   1:L PR[91] R[100]mm/sec CNT100;
   1:  PR[91,1] = PR[90,1] + -29.183;
   1:  PR[91,2] = PR[90,2] + 14.555;
   1:  PR[91,3] = PR[90,3] + 10.199;
   1:L PR[91] R[100]mm/sec CNT100;
   1:  PR[91,1] = PR[90,1] + -29.870;
   1:  PR[91,2] = PR[90,2] + 14.078;
   1:  PR[91,3] = PR[90,3] + 10.201;
   1:L PR[91] R[100]mm/sec CNT100;
   1:  PR[91,1] = PR[90,1] + -30.532;
   1:  PR[91,2] = PR[90,2] + 13.568;
   1:  PR[91,3] = PR[90,3] + 10.206;
   1:L PR[91] R[100]mm/sec CNT100;
   1:  PR[91,1] = PR[90,1] + -31.168;
   1:  PR[91,2] = PR[90,2] + 13.026;
   1:  PR[91,3] = PR[90,3] + 10.211;
   1:L PR[91] R[100]mm/sec CNT100;
   1:  PR[91,1] = PR[90,1] + -31.777;
   1:  PR[91,2] = PR[90,2] + 12.454;
   1:  PR[91,3] = PR[90,3] + 10.217;
   1:L PR[91] R[100]mm/sec CNT100;
   1:  PR[91,1] = PR[90,1] + -32.357;
   1:  PR[91,2] = PR[90,2] + 11.852;
   1:  PR[91,3] = PR[90,3] + 10.222;
   1:L PR[91] R[100]mm/sec CNT100;
   1:  PR[91,1] = PR[90,1] + -32.907;
   1:  PR[91,2] = PR[90,2] + 11.222;
   1:  PR[91,3] = PR[90,3] + 10.227;
   1:L PR[91] R[100]mm/sec CNT100;
   1:  PR[91,1] = PR[90,1] + -33.426;
   1:  PR[91,2] = PR[90,2] + 10.565;
   1:  PR[91,3] = PR[90,3] + 10.232;
   1:L PR[91] R[100]mm/sec CNT100;
   1:  PR[91,1] = PR[90,1] + -33.911;
   1:  PR[91,2] = PR[90,2] + 9.884;
   1:  PR[91,3] = PR[90,3] + 10.237;
   1:L PR[91] R[100]mm/sec CNT100;
   1:  PR[91,1] = PR[90,1] + -34.362;
   1:  PR[91,2] = PR[90,2] + 9.178;
   1:  PR[91,3] = PR[90,3] + 10.243;
   1:L PR[91] R[100]mm/sec CNT100;
   1:  PR[91,1] = PR[90,1] + -34.778;
   1:  PR[91,2] = PR[90,2] + 8.451;
   1:  PR[91,3] = PR[90,3] + 10.248;
   1:L PR[91] R[100]mm/sec CNT100;
   1:  PR[91,1] = PR[90,1] + -35.158;
   1:  PR[91,2] = PR[90,2] + 7.705;
   1:  PR[91,3] = PR[90,3] + 10.253;
   1:L PR[91] R[100]mm/sec CNT100;
   1:  PR[91,1] = PR[90,1] + -35.500;
   1:  PR[91,2] = PR[90,2] + 6.942;
   1:  PR[91,3] = PR[90,3] + 10.258;
   1:L PR[91] R[100]mm/sec CNT100;
   1:  PR[91,1] = PR[90,1] + -35.805;
   1:  PR[91,2] = PR[90,2] + 6.164;
   1:  PR[91,3] = PR[90,3] + 10.263;
   1:L PR[91] R[100]mm/sec CNT100;
   1:  PR[91,1] = PR[90,1] + -36.070;
   1:  PR[91,2] = PR[90,2] + 5.374;
   1:  PR[91,3] = PR[90,3] + 10.269;
   1:L PR[91] R[100]mm/sec CNT100;
   1:  PR[91,1] = PR[90,1] + -36.295;
   1:  PR[91,2] = PR[90,2] + 4.572;
   1:  PR[91,3] = PR[90,3] + 10.274;
   1:L PR[91] R[100]mm/sec CNT100;
   1:  PR[91,1] = PR[90,1] + -36.480;
   1:  PR[91,2] = PR[90,2] + 3.761;
   1:  PR[91,3] = PR[90,3] + 10.279;
   1:L PR[91] R[100]mm/sec CNT100;
   1:  PR[91,1] = PR[90,1] + -36.625;
   1:  PR[91,2] = PR[90,2] + 2.940;
   1:  PR[91,3] = PR[90,3] + 10.284;
   1:L PR[91] R[100]mm/sec CNT100;
   1:  PR[91,1] = PR[90,1] + -36.728;
   1:  PR[91,2] = PR[90,2] + 2.111;
   1:  PR[91,3] = PR[90,3] + 10.289;
   1:L PR[91] R[100]mm/sec CNT100;
   1:  PR[91,1] = PR[90,1] + -36.791;
   1:  PR[91,2] = PR[90,2] + 1.273;
   1:  PR[91,3] = PR[90,3] + 10.295;
   1:L PR[91] R[100]mm/sec CNT100;
   1:  PR[91,1] = PR[90,1] + -36.812;
   1:  PR[91,2] = PR[90,2] + 0.428;
   1:  PR[91,3] = PR[90,3] + 10.300;
   1:L PR[91] R[100]mm/sec CNT100;
   1:  PR[91,1] = PR[90,1] + -36.791;
   1:  PR[91,2] = PR[90,2] + -0.418;
   1:  PR[91,3] = PR[90,3] + 10.305;
   1:L PR[91] R[100]mm/sec CNT100;
   1:  PR[91,1] = PR[90,1] + -36.728;
   1:  PR[91,2] = PR[90,2] + -1.256;
   1:  PR[91,3] = PR[90,3] + 10.310;
   1:L PR[91] R[100]mm/sec CNT100;
   1:  PR[91,1] = PR[90,1] + -36.625;
   1:  PR[91,2] = PR[90,2] + -2.085;
   1:  PR[91,3] = PR[90,3] + 10.316;
   1:L PR[91] R[100]mm/sec CNT100;
   1:  PR[91,1] = PR[90,1] + -36.480;
   1:  PR[91,2] = PR[90,2] + -2.906;
   1:  PR[91,3] = PR[90,3] + 10.321;
   1:L PR[91] R[100]mm/sec CNT100;
   1:  PR[91,1] = PR[90,1] + -36.295;
   1:  PR[91,2] = PR[90,2] + -3.717;
   1:  PR[91,3] = PR[90,3] + 10.326;
   1:L PR[91] R[100]mm/sec CNT100;
   1:  PR[91,1] = PR[90,1] + -36.070;
   1:  PR[91,2] = PR[90,2] + -4.519;
   1:  PR[91,3] = PR[90,3] + 10.331;
   1:L PR[91] R[100]mm/sec CNT100;
   1:  PR[91,1] = PR[90,1] + -35.805;
   1:  PR[91,2] = PR[90,2] + -5.309;
   1:  PR[91,3] = PR[90,3] + 10.336;
   1:L PR[91] R[100]mm/sec CNT100;
   1:  PR[91,1] = PR[90,1] + -35.500;
   1:  PR[91,2] = PR[90,2] + -6.087;
   1:  PR[91,3] = PR[90,3] + 10.341;
   1:L PR[91] R[100]mm/sec CNT100;
   1:  PR[91,1] = PR[90,1] + -35.158;
   1:  PR[91,2] = PR[90,2] + -6.850;
   1:  PR[91,3] = PR[90,3] + 10.347;
   1:L PR[91] R[100]mm/sec CNT100;
   1:  PR[91,1] = PR[90,1] + -34.778;
   1:  PR[91,2] = PR[90,2] + -7.596;
   1:  PR[91,3] = PR[90,3] + 10.352;
   1:L PR[91] R[100]mm/sec CNT100;
   1:  PR[91,1] = PR[90,1] + -34.362;
   1:  PR[91,2] = PR[90,2] + -8.323;
   1:  PR[91,3] = PR[90,3] + 10.357;
   1:L PR[91] R[100]mm/sec CNT100;
   1:  PR[91,1] = PR[90,1] + -33.911;
   1:  PR[91,2] = PR[90,2] + -9.028;
   1:  PR[91,3] = PR[90,3] + 10.362;
   1:L PR[91] R[100]mm/sec CNT100;
   1:  PR[91,1] = PR[90,1] + -33.426;
   1:  PR[91,2] = PR[90,2] + -9.710;
   1:  PR[91,3] = PR[90,3] + 10.367;
   1:L PR[91] R[100]mm/sec CNT100;
   1:  PR[91,1] = PR[90,1] + -32.907;
   1:  PR[91,2] = PR[90,2] + -10.367;
   1:  PR[91,3] = PR[90,3] + 10.373;
   1:L PR[91] R[100]mm/sec CNT100;
   1:  PR[91,1] = PR[90,1] + -32.357;
   1:  PR[91,2] = PR[90,2] + -10.997;
   1:  PR[91,3] = PR[90,3] + 10.378;
   1:L PR[91] R[100]mm/sec CNT100;
   1:  PR[91,1] = PR[90,1] + -31.777;
   1:  PR[91,2] = PR[90,2] + -11.599;
   1:  PR[91,3] = PR[90,3] + 10.383;
   1:L PR[91] R[100]mm/sec CNT100;
   1:  PR[91,1] = PR[90,1] + -31.168;
   1:  PR[91,2] = PR[90,2] + -12.171;
   1:  PR[91,3] = PR[90,3] + 10.388;
   1:L PR[91] R[100]mm/sec CNT100;
   1:  PR[91,1] = PR[90,1] + -30.532;
   1:  PR[91,2] = PR[90,2] + -12.713;
   1:  PR[91,3] = PR[90,3] + 10.393;
   1:L PR[91] R[100]mm/sec CNT100;
   1:  PR[91,1] = PR[90,1] + -29.869;
   1:  PR[91,2] = PR[90,2] + -13.223;
   1:  PR[91,3] = PR[90,3] + 10.399;
   1:L PR[91] R[100]mm/sec CNT100;
   1:  PR[91,1] = PR[90,1] + -29.571;
   1:  PR[91,2] = PR[90,2] + -13.432;
   1:  PR[91,3] = PR[90,3] + 10.404;
   1:L PR[91] R[100]mm/sec CNT100;
   1:  PR[91,1] = PR[90,1] + -29.184;
   1:  PR[91,2] = PR[90,2] + -13.699;
   1:  PR[91,3] = PR[90,3] + 10.406;
   1:L PR[91] R[100]mm/sec CNT100;
   1:  PR[91,1] = PR[90,1] + -28.475;
   1:  PR[91,2] = PR[90,2] + -14.142;
   1:  PR[91,3] = PR[90,3] + 10.409;
   1:L PR[91] R[100]mm/sec CNT100;
   1:  PR[91,1] = PR[90,1] + -27.746;
   1:  PR[91,2] = PR[90,2] + -14.550;
   1:  PR[91,3] = PR[90,3] + 10.414;
   1:L PR[91] R[100]mm/sec CNT100;
   1:  PR[91,1] = PR[90,1] + -27.316;
   1:  PR[91,2] = PR[90,2] + -14.765;
   1:  PR[91,3] = PR[90,3] + 10.419;
   1:L PR[91] R[100]mm/sec CNT100;
   1:  PR[91,1] = PR[90,1] + -26.999;
   1:  PR[91,2] = PR[90,2] + -14.921;
   1:  PR[91,3] = PR[90,3] + 10.422;
   1:L PR[91] R[100]mm/sec CNT100;
   1:  PR[91,1] = PR[90,1] + -26.234;
   1:  PR[91,2] = PR[90,2] + -15.256;
   1:  PR[91,3] = PR[90,3] + 10.425;
   1:L PR[91] R[100]mm/sec CNT100;
   1:  PR[91,1] = PR[90,1] + -25.453;
   1:  PR[91,2] = PR[90,2] + -15.554;
   1:  PR[91,3] = PR[90,3] + 10.430;
   1:L PR[91] R[100]mm/sec CNT100;
   1:  PR[91,1] = PR[90,1] + -24.883;
   1:  PR[91,2] = PR[90,2] + -15.741;
   1:  PR[91,3] = PR[90,3] + 10.435;
   1:L PR[91] R[100]mm/sec CNT100;
   1:  PR[91,1] = PR[90,1] + -23.854;
   1:  PR[91,2] = PR[90,2] + -16.033;
   1:  PR[91,3] = PR[90,3] + 10.439;
   1:L PR[91] R[100]mm/sec CNT100;
   1:  PR[91,1] = PR[90,1] + -23.043;
   1:  PR[91,2] = PR[90,2] + -16.213;
   1:  PR[91,3] = PR[90,3] + 10.445;
   1:L PR[91] R[100]mm/sec CNT100;
   1:  PR[91,1] = PR[90,1] + -22.223;
   1:  PR[91,2] = PR[90,2] + -16.354;
   1:  PR[91,3] = PR[90,3] + 10.451;
   1:L PR[91] R[100]mm/sec CNT100;
   1:  PR[91,1] = PR[90,1] + -21.397;
   1:  PR[91,2] = PR[90,2] + -16.455;
   1:  PR[91,3] = PR[90,3] + 10.456;
   1:L PR[91] R[100]mm/sec CNT100;
   1:  PR[91,1] = PR[90,1] + -20.560;
   1:  PR[91,2] = PR[90,2] + -16.517;
   1:  PR[91,3] = PR[90,3] + 10.461;
   1:L PR[91] R[100]mm/sec CNT100;
   1:  PR[91,1] = PR[90,1] + -19.711;
   1:  PR[91,2] = PR[90,2] + -16.538;
   1:  PR[91,3] = PR[90,3] + 10.466;
   1:L PR[91] R[100]mm/sec CNT100;
   1:  PR[91,1] = PR[90,1] + -18.860;
   1:  PR[91,2] = PR[90,2] + -16.518;
   1:  PR[91,3] = PR[90,3] + 10.471;
   1:L PR[91] R[100]mm/sec CNT100;
   1:  PR[91,1] = PR[90,1] + -18.010;
   1:  PR[91,2] = PR[90,2] + -16.456;
   1:  PR[91,3] = PR[90,3] + 10.477;
   1:L PR[91] R[100]mm/sec CNT100;
   1:  PR[91,1] = PR[90,1] + -17.397;
   1:  PR[91,2] = PR[90,2] + -16.381;
   1:  PR[91,3] = PR[90,3] + 10.482;
   1:L PR[91] R[100]mm/sec CNT100;
   1:  PR[91,1] = PR[90,1] + -16.320;
   1:  PR[91,2] = PR[90,2] + -16.206;
   1:  PR[91,3] = PR[90,3] + 10.486;
   1:L PR[91] R[100]mm/sec CNT100;
   1:  PR[91,1] = PR[90,1] + -15.489;
   1:  PR[91,2] = PR[90,2] + -16.020;
   1:  PR[91,3] = PR[90,3] + 10.493;
   1:L PR[91] R[100]mm/sec CNT100;
   1:  PR[91,1] = PR[90,1] + -15.048;
   1:  PR[91,2] = PR[90,2] + -15.900;
   1:  PR[91,3] = PR[90,3] + 10.498;
   1:L PR[91] R[100]mm/sec CNT100;
   1:  PR[91,1] = PR[90,1] + -14.666;
   1:  PR[91,2] = PR[90,2] + -15.793;
   1:  PR[91,3] = PR[90,3] + 10.501;
   1:L PR[91] R[100]mm/sec CNT100;
   1:  PR[91,1] = PR[90,1] + -13.853;
   1:  PR[91,2] = PR[90,2] + -15.525;
   1:  PR[91,3] = PR[90,3] + 10.503;
   1:L PR[91] R[100]mm/sec CNT100;
   1:  PR[91,1] = PR[90,1] + -13.057;
   1:  PR[91,2] = PR[90,2] + -15.217;
   1:  PR[91,3] = PR[90,3] + 10.509;
   1:L PR[91] R[100]mm/sec CNT100;
   1:  PR[91,1] = PR[90,1] + -12.067;
   1:  PR[91,2] = PR[90,2] + -14.767;
   1:  PR[91,3] = PR[90,3] + 10.514;
   1:L PR[91] R[100]mm/sec CNT100;
   1:  PR[91,1] = PR[90,1] + -11.507;
   1:  PR[91,2] = PR[90,2] + -14.484;
   1:  PR[91,3] = PR[90,3] + 10.521;
   1:L PR[91] R[100]mm/sec CNT100;
   1:  PR[91,1] = PR[90,1] + -10.761;
   1:  PR[91,2] = PR[90,2] + -14.060;
   1:  PR[91,3] = PR[90,3] + 10.525;
   1:L PR[91] R[100]mm/sec CNT100;
   1:  PR[91,1] = PR[90,1] + -10.036;
   1:  PR[91,2] = PR[90,2] + -13.601;
   1:  PR[91,3] = PR[90,3] + 10.530;
   1:L PR[91] R[100]mm/sec CNT100;
   1:  PR[91,1] = PR[90,1] + -9.333;
   1:  PR[91,2] = PR[90,2] + -13.104;
   1:  PR[91,3] = PR[90,3] + 10.535;
   1:L PR[91] R[100]mm/sec CNT100;
   1:  PR[91,1] = PR[90,1] + -8.700;
   1:  PR[91,2] = PR[90,2] + -12.611;
   1:  PR[91,3] = PR[90,3] + 10.541;
   1:L PR[91] R[100]mm/sec CNT100;
   1:  PR[91,1] = PR[90,1] + -7.989;
   1:  PR[91,2] = PR[90,2] + -11.996;
   1:  PR[91,3] = PR[90,3] + 10.546;
   1:L PR[91] R[100]mm/sec CNT100;
   1:  PR[91,1] = PR[90,1] + -7.362;
   1:  PR[91,2] = PR[90,2] + -11.395;
   1:  PR[91,3] = PR[90,3] + 10.551;
   1:L PR[91] R[100]mm/sec CNT100;
   1:  PR[91,1] = PR[90,1] + -6.934;
   1:  PR[91,2] = PR[90,2] + -10.944;
   1:  PR[91,3] = PR[90,3] + 10.557;
   1:L PR[91] R[100]mm/sec CNT100;
   1:  PR[91,1] = PR[90,1] + -6.211;
   1:  PR[91,2] = PR[90,2] + -10.106;
   1:  PR[91,3] = PR[90,3] + 10.561;
   1:L PR[91] R[100]mm/sec CNT100;
   1:  PR[91,1] = PR[90,1] + -5.689;
   1:  PR[91,2] = PR[90,2] + -9.423;
   1:  PR[91,3] = PR[90,3] + 10.568;
   1:L PR[91] R[100]mm/sec CNT100;
   1:  PR[91,1] = PR[90,1] + -5.420;
   1:  PR[91,2] = PR[90,2] + -9.037;
   1:  PR[91,3] = PR[90,3] + 10.573;
   1:L PR[91] R[100]mm/sec CNT100;
   1:  PR[91,1] = PR[90,1] + -5.206;
   1:  PR[91,2] = PR[90,2] + -8.720;
   1:  PR[91,3] = PR[90,3] + 10.576;
   1:L PR[91] R[100]mm/sec CNT100;
   1:  PR[91,1] = PR[90,1] + -4.756;
   1:  PR[91,2] = PR[90,2] + -7.988;
   1:  PR[91,3] = PR[90,3] + 10.578;
   1:L PR[91] R[100]mm/sec CNT100;
   1:  PR[91,1] = PR[90,1] + -4.347;
   1:  PR[91,2] = PR[90,2] + -7.242;
   1:  PR[91,3] = PR[90,3] + 10.584;
   1:L PR[91] R[100]mm/sec CNT100;
   1:  PR[91,1] = PR[90,1] + -3.852;
   1:  PR[91,2] = PR[90,2] + -6.194;
   1:  PR[91,3] = PR[90,3] + 10.589;
   1:L PR[91] R[100]mm/sec CNT100;
   1:  PR[91,1] = PR[90,1] + -3.644;
   1:  PR[91,2] = PR[90,2] + -5.699;
   1:  PR[91,3] = PR[90,3] + 10.596;
   1:L PR[91] R[100]mm/sec CNT100;
   1:  PR[91,1] = PR[90,1] + -3.353;
   1:  PR[91,2] = PR[90,2] + -4.913;
   1:  PR[91,3] = PR[90,3] + 10.599;
   1:L PR[91] R[100]mm/sec CNT100;
   1:  PR[91,1] = PR[90,1] + -2.918;
   1:  PR[91,2] = PR[90,2] + -3.507;
   1:  PR[91,3] = PR[90,3] + 10.605;
   1:L PR[91] R[100]mm/sec CNT100;
   1:  PR[91,1] = PR[90,1] + -2.749;
   1:  PR[91,2] = PR[90,2] + -3.116;
   1:  PR[91,3] = PR[90,3] + 10.614;
   1:L PR[91] R[100]mm/sec CNT100;
   1:  PR[91,1] = PR[90,1] + -2.607;
   1:  PR[91,2] = PR[90,2] + -2.852;
   1:  PR[91,3] = PR[90,3] + 10.616;
   1:L PR[91] R[100]mm/sec CNT100;
   1:  PR[91,1] = PR[90,1] + -2.339;
   1:  PR[91,2] = PR[90,2] + -2.452;
   1:  PR[91,3] = PR[90,3] + 10.618;
   1:L PR[91] R[100]mm/sec CNT100;
   1:  PR[91,1] = PR[90,1] + -2.023;
   1:  PR[91,2] = PR[90,2] + -2.095;
   1:  PR[91,3] = PR[90,3] + 10.621;
   1:L PR[91] R[100]mm/sec CNT100;
   1:  PR[91,1] = PR[90,1] + -1.688;
   1:  PR[91,2] = PR[90,2] + -1.805;
   1:  PR[91,3] = PR[90,3] + 10.624;
   1:L PR[91] R[100]mm/sec CNT100;
   1:  PR[91,1] = PR[90,1] + -1.335;
   1:  PR[91,2] = PR[90,2] + -1.579;
   1:  PR[91,3] = PR[90,3] + 10.627;
   1:L PR[91] R[100]mm/sec CNT100;
   1:  PR[91,1] = PR[90,1] + -0.967;
   1:  PR[91,2] = PR[90,2] + -1.413;
   1:  PR[91,3] = PR[90,3] + 10.630;
   1:L PR[91] R[100]mm/sec CNT100;
   1:  PR[91,1] = PR[90,1] + -0.512;
   1:  PR[91,2] = PR[90,2] + -1.295;
   1:  PR[91,3] = PR[90,3] + 10.632;
   1:L PR[91] R[100]mm/sec CNT100;
   1:  PR[91,1] = PR[90,1] + -0.120;
   1:  PR[91,2] = PR[90,2] + -1.263;
   1:  PR[91,3] = PR[90,3] + 10.635;
   1:L PR[91] R[100]mm/sec CNT100;
   1:  PR[91,1] = PR[90,1] + 0.273;
   1:  PR[91,2] = PR[90,2] + -1.295;
   1:  PR[91,3] = PR[90,3] + 10.638;
   1:L PR[91] R[100]mm/sec CNT100;
   1:  PR[91] = PR[90];
   1:  PR[91,1] = PR[90,1] + 0.506;
   1:  PR[91,2] = PR[90,2] + -2.523;
   1:  PR[91,3] = PR[90,3] + 11.970;
   1:L PR[91] R[100]mm/sec CNT100;
   1:  PR[91,1] = PR[90,1] + 0.886;
   1:  PR[91,2] = PR[90,2] + -2.652;
   1:  PR[91,3] = PR[90,3] + 10.643;
   1:L PR[91] R[100]mm/sec CNT100;
   1:  PR[91,1] = PR[90,1] + 1.255;
   1:  PR[91,2] = PR[90,2] + -2.842;
   1:  PR[91,3] = PR[90,3] + 10.645;
   1:L PR[91] R[100]mm/sec CNT100;
   1:  PR[91,1] = PR[90,1] + 1.659;
   1:  PR[91,2] = PR[90,2] + -3.142;
   1:  PR[91,3] = PR[90,3] + 10.648;
   1:L PR[91] R[100]mm/sec CNT100;
   1:  PR[91,1] = PR[90,1] + 1.889;
   1:  PR[91,2] = PR[90,2] + -3.364;
   1:  PR[91,3] = PR[90,3] + 10.651;
   1:L PR[91] R[100]mm/sec CNT100;
   1:  PR[91,1] = PR[90,1] + 2.154;
   1:  PR[91,2] = PR[90,2] + -3.679;
   1:  PR[91,3] = PR[90,3] + 10.653;
   1:L PR[91] R[100]mm/sec CNT100;
   1:  PR[91,1] = PR[90,1] + 2.385;
   1:  PR[91,2] = PR[90,2] + -4.031;
   1:  PR[91,3] = PR[90,3] + 10.656;
   1:L PR[91] R[100]mm/sec CNT100;
   1:  PR[91,1] = PR[90,1] + 2.583;
   1:  PR[91,2] = PR[90,2] + -4.414;
   1:  PR[91,3] = PR[90,3] + 10.658;
   1:L PR[91] R[100]mm/sec CNT100;
   1:  PR[91,1] = PR[90,1] + 2.949;
   1:  PR[91,2] = PR[90,2] + -5.405;
   1:  PR[91,3] = PR[90,3] + 10.661;
   1:L PR[91] R[100]mm/sec CNT100;
   1:  PR[91,1] = PR[90,1] + 3.271;
   1:  PR[91,2] = PR[90,2] + -6.190;
   1:  PR[91,3] = PR[90,3] + 10.668;
   1:L PR[91] R[100]mm/sec CNT100;
   1:  PR[91,1] = PR[90,1] + 3.632;
   1:  PR[91,2] = PR[90,2] + -6.960;
   1:  PR[91,3] = PR[90,3] + 10.673;
   1:L PR[91] R[100]mm/sec CNT100;
   1:  PR[91,1] = PR[90,1] + 4.033;
   1:  PR[91,2] = PR[90,2] + -7.716;
   1:  PR[91,3] = PR[90,3] + 10.679;
   1:L PR[91] R[100]mm/sec CNT100;
   1:  PR[91,1] = PR[90,1] + 4.471;
   1:  PR[91,2] = PR[90,2] + -8.454;
   1:  PR[91,3] = PR[90,3] + 10.684;
   1:L PR[91] R[100]mm/sec CNT100;
   1:  PR[91,1] = PR[90,1] + 4.945;
   1:  PR[91,2] = PR[90,2] + -9.170;
   1:  PR[91,3] = PR[90,3] + 10.689;
   1:L PR[91] R[100]mm/sec CNT100;
   1:  PR[91,1] = PR[90,1] + 5.455;
   1:  PR[91,2] = PR[90,2] + -9.862;
   1:  PR[91,3] = PR[90,3] + 10.695;
   1:L PR[91] R[100]mm/sec CNT100;
   1:  PR[91,1] = PR[90,1] + 5.998;
   1:  PR[91,2] = PR[90,2] + -10.527;
   1:  PR[91,3] = PR[90,3] + 10.700;
   1:L PR[91] R[100]mm/sec CNT100;
   1:  PR[91,1] = PR[90,1] + 6.575;
   1:  PR[91,2] = PR[90,2] + -11.165;
   1:  PR[91,3] = PR[90,3] + 10.706;
   1:L PR[91] R[100]mm/sec CNT100;
   1:  PR[91,1] = PR[90,1] + 6.949;
   1:  PR[91,2] = PR[90,2] + -11.541;
   1:  PR[91,3] = PR[90,3] + 10.711;
   1:L PR[91] R[100]mm/sec CNT100;
   1:  PR[91,1] = PR[90,1] + 7.181;
   1:  PR[91,2] = PR[90,2] + -11.769;
   1:  PR[91,3] = PR[90,3] + 10.715;
   1:L PR[91] R[100]mm/sec CNT100;
   1:  PR[91,1] = PR[90,1] + 7.820;
   1:  PR[91,2] = PR[90,2] + -12.345;
   1:  PR[91,3] = PR[90,3] + 10.717;
   1:L PR[91] R[100]mm/sec CNT100;
   1:  PR[91,1] = PR[90,1] + 8.486;
   1:  PR[91,2] = PR[90,2] + -12.889;
   1:  PR[91,3] = PR[90,3] + 10.722;
   1:L PR[91] R[100]mm/sec CNT100;
   1:  PR[91,1] = PR[90,1] + 8.743;
   1:  PR[91,2] = PR[90,2] + -13.080;
   1:  PR[91,3] = PR[90,3] + 10.727;
   1:L PR[91] R[100]mm/sec CNT100;
   1:  PR[91,1] = PR[90,1] + 9.176;
   1:  PR[91,2] = PR[90,2] + -13.396;
   1:  PR[91,3] = PR[90,3] + 10.730;
   1:L PR[91] R[100]mm/sec CNT100;
   1:  PR[91,1] = PR[90,1] + 9.892;
   1:  PR[91,2] = PR[90,2] + -13.870;
   1:  PR[91,3] = PR[90,3] + 10.733;
   1:L PR[91] R[100]mm/sec CNT100;
   1:  PR[91,1] = PR[90,1] + 10.630;
   1:  PR[91,2] = PR[90,2] + -14.309;
   1:  PR[91,3] = PR[90,3] + 10.738;
   1:L PR[91] R[100]mm/sec CNT100;
   1:  PR[91,1] = PR[90,1] + 11.389;
   1:  PR[91,2] = PR[90,2] + -14.711;
   1:  PR[91,3] = PR[90,3] + 10.744;
   1:L PR[91] R[100]mm/sec CNT100;
   1:  PR[91,1] = PR[90,1] + 12.175;
   1:  PR[91,2] = PR[90,2] + -15.079;
   1:  PR[91,3] = PR[90,3] + 10.749;
   1:L PR[91] R[100]mm/sec CNT100;
   1:  PR[91,1] = PR[90,1] + 12.890;
   1:  PR[91,2] = PR[90,2] + -15.375;
   1:  PR[91,3] = PR[90,3] + 10.755;
   1:L PR[91] R[100]mm/sec CNT100;
   1:  PR[91,1] = PR[90,1] + 13.651;
   1:  PR[91,2] = PR[90,2] + -15.651;
   1:  PR[91,3] = PR[90,3] + 10.760;
   1:L PR[91] R[100]mm/sec CNT100;
   1:  PR[91,1] = PR[90,1] + 14.424;
   1:  PR[91,2] = PR[90,2] + -15.892;
   1:  PR[91,3] = PR[90,3] + 10.765;
   1:L PR[91] R[100]mm/sec CNT100;
   1:  PR[91,1] = PR[90,1] + 15.210;
   1:  PR[91,2] = PR[90,2] + -16.097;
   1:  PR[91,3] = PR[90,3] + 10.770;
   1:L PR[91] R[100]mm/sec CNT100;
   1:  PR[91,1] = PR[90,1] + 16.007;
   1:  PR[91,2] = PR[90,2] + -16.267;
   1:  PR[91,3] = PR[90,3] + 10.775;
   1:L PR[91] R[100]mm/sec CNT100;
   1:  PR[91,1] = PR[90,1] + 16.813;
   1:  PR[91,2] = PR[90,2] + -16.399;
   1:  PR[91,3] = PR[90,3] + 10.780;
   1:L PR[91] R[100]mm/sec CNT100;
   1:  PR[91,1] = PR[90,1] + 17.626;
   1:  PR[91,2] = PR[90,2] + -16.495;
   1:  PR[91,3] = PR[90,3] + 10.785;
   1:L PR[91] R[100]mm/sec CNT100;
   1:  PR[91,1] = PR[90,1] + 18.444;
   1:  PR[91,2] = PR[90,2] + -16.552;
   1:  PR[91,3] = PR[90,3] + 10.791;
   1:L PR[91] R[100]mm/sec CNT100;
   1:  PR[91,1] = PR[90,1] + 19.266;
   1:  PR[91,2] = PR[90,2] + -16.571;
   1:  PR[91,3] = PR[90,3] + 10.796;
   1:L PR[91] R[100]mm/sec CNT100;
   1:  PR[91,1] = PR[90,1] + 20.090;
   1:  PR[91,2] = PR[90,2] + -16.551;
   1:  PR[91,3] = PR[90,3] + 10.801;
   1:L PR[91] R[100]mm/sec CNT100;
   1:  PR[91,1] = PR[90,1] + 20.914;
   1:  PR[91,2] = PR[90,2] + -16.493;
   1:  PR[91,3] = PR[90,3] + 10.806;
   1:L PR[91] R[100]mm/sec CNT100;
   1:  PR[91,1] = PR[90,1] + 21.736;
   1:  PR[91,2] = PR[90,2] + -16.395;
   1:  PR[91,3] = PR[90,3] + 10.811;
   1:L PR[91] R[100]mm/sec CNT100;
   1:  PR[91,1] = PR[90,1] + 22.576;
   1:  PR[91,2] = PR[90,2] + -16.254;
   1:  PR[91,3] = PR[90,3] + 10.817;
   1:L PR[91] R[100]mm/sec CNT100;
   1:  PR[91,1] = PR[90,1] + 23.410;
   1:  PR[91,2] = PR[90,2] + -16.072;
   1:  PR[91,3] = PR[90,3] + 10.822;
   1:L PR[91] R[100]mm/sec CNT100;
   1:  PR[91,1] = PR[90,1] + 24.233;
   1:  PR[91,2] = PR[90,2] + -15.849;
   1:  PR[91,3] = PR[90,3] + 10.827;
   1:L PR[91] R[100]mm/sec CNT100;
   1:  PR[91,1] = PR[90,1] + 25.043;
   1:  PR[91,2] = PR[90,2] + -15.586;
   1:  PR[91,3] = PR[90,3] + 10.833;
   1:L PR[91] R[100]mm/sec CNT100;
   1:  PR[91,1] = PR[90,1] + 25.838;
   1:  PR[91,2] = PR[90,2] + -15.284;
   1:  PR[91,3] = PR[90,3] + 10.838;
   1:L PR[91] R[100]mm/sec CNT100;
   1:  PR[91,1] = PR[90,1] + 26.617;
   1:  PR[91,2] = PR[90,2] + -14.945;
   1:  PR[91,3] = PR[90,3] + 10.844;
   1:L PR[91] R[100]mm/sec CNT100;
   1:  PR[91,1] = PR[90,1] + 27.376;
   1:  PR[91,2] = PR[90,2] + -14.568;
   1:  PR[91,3] = PR[90,3] + 10.849;
   1:L PR[91] R[100]mm/sec CNT100;
   1:  PR[91,1] = PR[90,1] + 28.115;
   1:  PR[91,2] = PR[90,2] + -14.155;
   1:  PR[91,3] = PR[90,3] + 10.854;
   1:L PR[91] R[100]mm/sec CNT100;
   1:  PR[91,1] = PR[90,1] + 28.832;
   1:  PR[91,2] = PR[90,2] + -13.707;
   1:  PR[91,3] = PR[90,3] + 10.860;
   1:L PR[91] R[100]mm/sec CNT100;
   1:  PR[91,1] = PR[90,1] + 29.525;
   1:  PR[91,2] = PR[90,2] + -13.225;
   1:  PR[91,3] = PR[90,3] + 10.865;
   1:L PR[91] R[100]mm/sec CNT100;
   1:  PR[91,1] = PR[90,1] + 30.193;
   1:  PR[91,2] = PR[90,2] + -12.710;
   1:  PR[91,3] = PR[90,3] + 10.870;
   1:L PR[91] R[100]mm/sec CNT100;
   1:  PR[91,1] = PR[90,1] + 30.833;
   1:  PR[91,2] = PR[90,2] + -12.163;
   1:  PR[91,3] = PR[90,3] + 10.876;
   1:L PR[91] R[100]mm/sec CNT100;
   1:  PR[91,1] = PR[90,1] + 31.445;
   1:  PR[91,2] = PR[90,2] + -11.586;
   1:  PR[91,3] = PR[90,3] + 10.881;
   1:L PR[91] R[100]mm/sec CNT100;
   1:  PR[91,1] = PR[90,1] + 32.027;
   1:  PR[91,2] = PR[90,2] + -10.980;
   1:  PR[91,3] = PR[90,3] + 10.886;
   1:L PR[91] R[100]mm/sec CNT100;
   1:  PR[91,1] = PR[90,1] + 32.578;
   1:  PR[91,2] = PR[90,2] + -10.346;
   1:  PR[91,3] = PR[90,3] + 10.892;
   1:L PR[91] R[100]mm/sec CNT100;
   1:  PR[91,1] = PR[90,1] + 33.097;
   1:  PR[91,2] = PR[90,2] + -9.685;
   1:  PR[91,3] = PR[90,3] + 10.897;
   1:L PR[91] R[100]mm/sec CNT100;
   1:  PR[91,1] = PR[90,1] + 33.582;
   1:  PR[91,2] = PR[90,2] + -9.001;
   1:  PR[91,3] = PR[90,3] + 10.902;
   1:L PR[91] R[100]mm/sec CNT100;
   1:  PR[91,1] = PR[90,1] + 34.033;
   1:  PR[91,2] = PR[90,2] + -8.294;
   1:  PR[91,3] = PR[90,3] + 10.908;
   1:L PR[91] R[100]mm/sec CNT100;
   1:  PR[91,1] = PR[90,1] + 34.448;
   1:  PR[91,2] = PR[90,2] + -7.567;
   1:  PR[91,3] = PR[90,3] + 10.913;
   1:L PR[91] R[100]mm/sec CNT100;
   1:  PR[91,1] = PR[90,1] + 34.826;
   1:  PR[91,2] = PR[90,2] + -6.822;
   1:  PR[91,3] = PR[90,3] + 10.918;
   1:L PR[91] R[100]mm/sec CNT100;
   1:  PR[91,1] = PR[90,1] + 35.167;
   1:  PR[91,2] = PR[90,2] + -6.061;
   1:  PR[91,3] = PR[90,3] + 10.924;
   1:L PR[91] R[100]mm/sec CNT100;
   1:  PR[91,1] = PR[90,1] + 35.476;
   1:  PR[91,2] = PR[90,2] + -5.270;
   1:  PR[91,3] = PR[90,3] + 10.929;
   1:L PR[91] R[100]mm/sec CNT100;
   1:  PR[91,1] = PR[90,1] + 35.735;
   1:  PR[91,2] = PR[90,2] + -4.497;
   1:  PR[91,3] = PR[90,3] + 10.934;
   1:L PR[91] R[100]mm/sec CNT100;
   1:  PR[91,1] = PR[90,1] + 35.958;
   1:  PR[91,2] = PR[90,2] + -3.701;
   1:  PR[91,3] = PR[90,3] + 10.940;
   1:L PR[91] R[100]mm/sec CNT100;
   1:  PR[91,1] = PR[90,1] + 36.143;
   1:  PR[91,2] = PR[90,2] + -2.885;
   1:  PR[91,3] = PR[90,3] + 10.945;
   1:L PR[91] R[100]mm/sec CNT100;
   1:  PR[91,1] = PR[90,1] + 36.283;
   1:  PR[91,2] = PR[90,2] + -2.083;
   1:  PR[91,3] = PR[90,3] + 10.950;
   1:L PR[91] R[100]mm/sec CNT100;
   1:  PR[91,1] = PR[90,1] + 36.386;
   1:  PR[91,2] = PR[90,2] + -1.256;
   1:  PR[91,3] = PR[90,3] + 10.955;
   1:L PR[91] R[100]mm/sec CNT100;
   1:  PR[91,1] = PR[90,1] + 36.448;
   1:  PR[91,2] = PR[90,2] + -0.419;
   1:  PR[91,3] = PR[90,3] + 10.960;
   1:L PR[91] R[100]mm/sec CNT100;
   1:  PR[91,1] = PR[90,1] + 36.468;
   1:  PR[91,2] = PR[90,2] + 0.428;
   1:  PR[91,3] = PR[90,3] + 10.966;
   1:L PR[91] R[100]mm/sec CNT100;
   1:  PR[91,1] = PR[90,1] + 36.448;
   1:  PR[91,2] = PR[90,2] + 1.274;
   1:  PR[91,3] = PR[90,3] + 10.971;
   1:L PR[91] R[100]mm/sec CNT100;
   1:  PR[91,1] = PR[90,1] + 36.386;
   1:  PR[91,2] = PR[90,2] + 2.111;
   1:  PR[91,3] = PR[90,3] + 10.977;
   1:L PR[91] R[100]mm/sec CNT100;
   1:  PR[91,1] = PR[90,1] + 36.283;
   1:  PR[91,2] = PR[90,2] + 2.938;
   1:  PR[91,3] = PR[90,3] + 10.982;
   1:L PR[91] R[100]mm/sec CNT100;
   1:  PR[91,1] = PR[90,1] + 36.140;
   1:  PR[91,2] = PR[90,2] + 3.755;
   1:  PR[91,3] = PR[90,3] + 10.987;
   1:L PR[91] R[100]mm/sec CNT100;
   1:  PR[91,1] = PR[90,1] + 35.957;
   1:  PR[91,2] = PR[90,2] + 4.561;
   1:  PR[91,3] = PR[90,3] + 10.992;
   1:L PR[91] R[100]mm/sec CNT100;
   1:  PR[91,1] = PR[90,1] + 35.733;
   1:  PR[91,2] = PR[90,2] + 5.357;
   1:  PR[91,3] = PR[90,3] + 10.998;
   1:L PR[91] R[100]mm/sec CNT100;
   1:  PR[91,1] = PR[90,1] + 35.470;
   1:  PR[91,2] = PR[90,2] + 6.143;
   1:  PR[91,3] = PR[90,3] + 11.003;
   1:L PR[91] R[100]mm/sec CNT100;
   1:  PR[91,1] = PR[90,1] + 35.167;
   1:  PR[91,2] = PR[90,2] + 6.916;
   1:  PR[91,3] = PR[90,3] + 11.008;
   1:L PR[91] R[100]mm/sec CNT100;
   1:  PR[91,1] = PR[90,1] + 34.826;
   1:  PR[91,2] = PR[90,2] + 7.677;
   1:  PR[91,3] = PR[90,3] + 11.013;
   1:L PR[91] R[100]mm/sec CNT100;
   1:  PR[91,1] = PR[90,1] + 34.448;
   1:  PR[91,2] = PR[90,2] + 8.422;
   1:  PR[91,3] = PR[90,3] + 11.019;
   1:L PR[91] R[100]mm/sec CNT100;
   1:  PR[91,1] = PR[90,1] + 34.033;
   1:  PR[91,2] = PR[90,2] + 9.149;
   1:  PR[91,3] = PR[90,3] + 11.024;
   1:L PR[91] R[100]mm/sec CNT100;
   1:  PR[91,1] = PR[90,1] + 33.582;
   1:  PR[91,2] = PR[90,2] + 9.856;
   1:  PR[91,3] = PR[90,3] + 11.029;
   1:L PR[91] R[100]mm/sec CNT100;
   1:  PR[91,1] = PR[90,1] + 33.097;
   1:  PR[91,2] = PR[90,2] + 10.540;
   1:  PR[91,3] = PR[90,3] + 11.035;
   1:L PR[91] R[100]mm/sec CNT100;
   1:  PR[91,1] = PR[90,1] + 32.578;
   1:  PR[91,2] = PR[90,2] + 11.201;
   1:  PR[91,3] = PR[90,3] + 11.040;
   1:L PR[91] R[100]mm/sec CNT100;
   1:  PR[91,1] = PR[90,1] + 32.027;
   1:  PR[91,2] = PR[90,2] + 11.835;
   1:  PR[91,3] = PR[90,3] + 11.045;
   1:L PR[91] R[100]mm/sec CNT100;
   1:  PR[91,1] = PR[90,1] + 31.445;
   1:  PR[91,2] = PR[90,2] + 12.441;
   1:  PR[91,3] = PR[90,3] + 11.051;
   1:L PR[91] R[100]mm/sec CNT100;
   1:  PR[91,1] = PR[90,1] + 30.833;
   1:  PR[91,2] = PR[90,2] + 13.018;
   1:  PR[91,3] = PR[90,3] + 11.056;
   1:L PR[91] R[100]mm/sec CNT100;
   1:  PR[91,1] = PR[90,1] + 30.193;
   1:  PR[91,2] = PR[90,2] + 13.565;
   1:  PR[91,3] = PR[90,3] + 11.061;
   1:L PR[91] R[100]mm/sec CNT100;
   1:  PR[91,1] = PR[90,1] + 29.525;
   1:  PR[91,2] = PR[90,2] + 14.080;
   1:  PR[91,3] = PR[90,3] + 11.067;
   1:L PR[91] R[100]mm/sec CNT100;
   1:  PR[91,1] = PR[90,1] + 28.832;
   1:  PR[91,2] = PR[90,2] + 14.562;
   1:  PR[91,3] = PR[90,3] + 11.072;
   1:L PR[91] R[100]mm/sec CNT100;
   1:  PR[91,1] = PR[90,1] + 28.115;
   1:  PR[91,2] = PR[90,2] + 15.010;
   1:  PR[91,3] = PR[90,3] + 11.077;
   1:L PR[91] R[100]mm/sec CNT100;
   1:  PR[91,1] = PR[90,1] + 27.771;
   1:  PR[91,2] = PR[90,2] + 15.204;
   1:  PR[91,3] = PR[90,3] + 11.083;
   1:L PR[91] R[100]mm/sec CNT100;
   1:  PR[91,1] = PR[90,1] + 27.377;
   1:  PR[91,2] = PR[90,2] + 15.423;
   1:  PR[91,3] = PR[90,3] + 11.085;
   1:L PR[91] R[100]mm/sec CNT100;
   1:  PR[91,1] = PR[90,1] + 26.617;
   1:  PR[91,2] = PR[90,2] + 15.800;
   1:  PR[91,3] = PR[90,3] + 11.088;
   1:L PR[91] R[100]mm/sec CNT100;
   1:  PR[91,1] = PR[90,1] + 25.838;
   1:  PR[91,2] = PR[90,2] + 16.139;
   1:  PR[91,3] = PR[90,3] + 11.093;
   1:L PR[91] R[100]mm/sec CNT100;
   1:  PR[91,1] = PR[90,1] + 25.043;
   1:  PR[91,2] = PR[90,2] + 16.441;
   1:  PR[91,3] = PR[90,3] + 11.099;
   1:L PR[91] R[100]mm/sec CNT100;
   1:  PR[91,1] = PR[90,1] + 24.233;
   1:  PR[91,2] = PR[90,2] + 16.704;
   1:  PR[91,3] = PR[90,3] + 11.104;
   1:L PR[91] R[100]mm/sec CNT100;
   1:  PR[91,1] = PR[90,1] + 23.410;
   1:  PR[91,2] = PR[90,2] + 16.927;
   1:  PR[91,3] = PR[90,3] + 11.109;
   1:L PR[91] R[100]mm/sec CNT100;
   1:  PR[91,1] = PR[90,1] + 22.576;
   1:  PR[91,2] = PR[90,2] + 17.110;
   1:  PR[91,3] = PR[90,3] + 11.115;
   1:L PR[91] R[100]mm/sec CNT100;
   1:  PR[91,1] = PR[90,1] + 21.727;
   1:  PR[91,2] = PR[90,2] + 17.252;
   1:  PR[91,3] = PR[90,3] + 11.120;
   1:L PR[91] R[100]mm/sec CNT100;
   1:  PR[91,1] = PR[90,1] + 20.914;
   1:  PR[91,2] = PR[90,2] + 17.348;
   1:  PR[91,3] = PR[90,3] + 11.126;
   1:L PR[91] R[100]mm/sec CNT100;
   1:  PR[91,1] = PR[90,1] + 20.090;
   1:  PR[91,2] = PR[90,2] + 17.406;
   1:  PR[91,3] = PR[90,3] + 11.131;
   1:L PR[91] R[100]mm/sec CNT100;
   1:  PR[91,1] = PR[90,1] + 19.266;
   1:  PR[91,2] = PR[90,2] + 17.426;
   1:  PR[91,3] = PR[90,3] + 11.136;
   1:L PR[91] R[100]mm/sec CNT100;
   1:  PR[91,1] = PR[90,1] + 18.444;
   1:  PR[91,2] = PR[90,2] + 17.407;
   1:  PR[91,3] = PR[90,3] + 11.141;
   1:L PR[91] R[100]mm/sec CNT100;
   1:  PR[91,1] = PR[90,1] + 17.626;
   1:  PR[91,2] = PR[90,2] + 17.350;
   1:  PR[91,3] = PR[90,3] + 11.147;
   1:L PR[91] R[100]mm/sec CNT100;
   1:  PR[91,1] = PR[90,1] + 16.813;
   1:  PR[91,2] = PR[90,2] + 17.255;
   1:  PR[91,3] = PR[90,3] + 11.152;
   1:L PR[91] R[100]mm/sec CNT100;
   1:  PR[91,1] = PR[90,1] + 16.007;
   1:  PR[91,2] = PR[90,2] + 17.122;
   1:  PR[91,3] = PR[90,3] + 11.157;
   1:L PR[91] R[100]mm/sec CNT100;
   1:  PR[91,1] = PR[90,1] + 15.210;
   1:  PR[91,2] = PR[90,2] + 16.952;
   1:  PR[91,3] = PR[90,3] + 11.162;
   1:L PR[91] R[100]mm/sec CNT100;
   1:  PR[91,1] = PR[90,1] + 14.424;
   1:  PR[91,2] = PR[90,2] + 16.747;
   1:  PR[91,3] = PR[90,3] + 11.167;
   1:L PR[91] R[100]mm/sec CNT100;
   1:  PR[91,1] = PR[90,1] + 13.651;
   1:  PR[91,2] = PR[90,2] + 16.506;
   1:  PR[91,3] = PR[90,3] + 11.172;
   1:L PR[91] R[100]mm/sec CNT100;
   1:  PR[91,1] = PR[90,1] + 12.890;
   1:  PR[91,2] = PR[90,2] + 16.230;
   1:  PR[91,3] = PR[90,3] + 11.178;
   1:L PR[91] R[100]mm/sec CNT100;
   1:  PR[91,1] = PR[90,1] + 12.145;
   1:  PR[91,2] = PR[90,2] + 15.921;
   1:  PR[91,3] = PR[90,3] + 11.183;
   1:L PR[91] R[100]mm/sec CNT100;
   1:  PR[91,1] = PR[90,1] + 11.389;
   1:  PR[91,2] = PR[90,2] + 15.566;
   1:  PR[91,3] = PR[90,3] + 11.188;
   1:L PR[91] R[100]mm/sec CNT100;
   1:  PR[91,1] = PR[90,1] + 10.630;
   1:  PR[91,2] = PR[90,2] + 15.164;
   1:  PR[91,3] = PR[90,3] + 11.193;
   1:L PR[91] R[100]mm/sec CNT100;
   1:  PR[91,1] = PR[90,1] + 9.891;
   1:  PR[91,2] = PR[90,2] + 14.725;
   1:  PR[91,3] = PR[90,3] + 11.199;
   1:L PR[91] R[100]mm/sec CNT100;
   1:  PR[91,1] = PR[90,1] + 9.392;
   1:  PR[91,2] = PR[90,2] + 14.396;
   1:  PR[91,3] = PR[90,3] + 11.204;
   1:L PR[91] R[100]mm/sec CNT100;
   1:  PR[91,1] = PR[90,1] + 8.482;
   1:  PR[91,2] = PR[90,2] + 13.741;
   1:  PR[91,3] = PR[90,3] + 11.208;
   1:L PR[91] R[100]mm/sec CNT100;
   1:  PR[91,1] = PR[90,1] + 7.820;
   1:  PR[91,2] = PR[90,2] + 13.200;
   1:  PR[91,3] = PR[90,3] + 11.215;
   1:L PR[91] R[100]mm/sec CNT100;
   1:  PR[91,1] = PR[90,1] + 7.184;
   1:  PR[91,2] = PR[90,2] + 12.627;
   1:  PR[91,3] = PR[90,3] + 11.220;
   1:L PR[91] R[100]mm/sec CNT100;
   1:  PR[91,1] = PR[90,1] + 6.393;
   1:  PR[91,2] = PR[90,2] + 11.821;
   1:  PR[91,3] = PR[90,3] + 11.226;
   1:L PR[91] R[100]mm/sec CNT100;
   1:  PR[91,1] = PR[90,1] + 5.999;
   1:  PR[91,2] = PR[90,2] + 11.383;
   1:  PR[91,3] = PR[90,3] + 11.233;
   1:L PR[91] R[100]mm/sec CNT100;
   1:  PR[91,1] = PR[90,1] + 5.455;
   1:  PR[91,2] = PR[90,2] + 10.717;
   1:  PR[91,3] = PR[90,3] + 11.237;
   1:L PR[91] R[100]mm/sec CNT100;
   1:  PR[91,1] = PR[90,1] + 4.946;
   1:  PR[91,2] = PR[90,2] + 10.025;
   1:  PR[91,3] = PR[90,3] + 11.242;
   1:L PR[91] R[100]mm/sec CNT100;
   1:  PR[91,1] = PR[90,1] + 4.459;
   1:  PR[91,2] = PR[90,2] + 9.288;
   1:  PR[91,3] = PR[90,3] + 11.248;
   1:L PR[91] R[100]mm/sec CNT100;
   1:  PR[91,1] = PR[90,1] + 4.033;
   1:  PR[91,2] = PR[90,2] + 8.571;
   1:  PR[91,3] = PR[90,3] + 11.253;
   1:L PR[91] R[100]mm/sec CNT100;
   1:  PR[91,1] = PR[90,1] + 3.632;
   1:  PR[91,2] = PR[90,2] + 7.815;
   1:  PR[91,3] = PR[90,3] + 11.258;
   1:L PR[91] R[100]mm/sec CNT100;
   1:  PR[91,1] = PR[90,1] + 3.271;
   1:  PR[91,2] = PR[90,2] + 7.045;
   1:  PR[91,3] = PR[90,3] + 11.264;
   1:L PR[91] R[100]mm/sec CNT100;
   1:  PR[91,1] = PR[90,1] + 2.948;
   1:  PR[91,2] = PR[90,2] + 6.260;
   1:  PR[91,3] = PR[90,3] + 11.269;
   1:L PR[91] R[100]mm/sec CNT100;
   1:  PR[91,1] = PR[90,1] + 2.582;
   1:  PR[91,2] = PR[90,2] + 5.269;
   1:  PR[91,3] = PR[90,3] + 11.275;
   1:L PR[91] R[100]mm/sec CNT100;
   1:  PR[91,1] = PR[90,1] + 2.385;
   1:  PR[91,2] = PR[90,2] + 4.885;
   1:  PR[91,3] = PR[90,3] + 11.281;
   1:L PR[91] R[100]mm/sec CNT100;
   1:  PR[91,1] = PR[90,1] + 2.153;
   1:  PR[91,2] = PR[90,2] + 4.534;
   1:  PR[91,3] = PR[90,3] + 11.284;
   1:L PR[91] R[100]mm/sec CNT100;
   1:  PR[91,1] = PR[90,1] + 1.886;
   1:  PR[91,2] = PR[90,2] + 4.215;
   1:  PR[91,3] = PR[90,3] + 11.287;
   1:L PR[91] R[100]mm/sec CNT100;
   1:  PR[91,1] = PR[90,1] + 1.585;
   1:  PR[91,2] = PR[90,2] + 3.933;
   1:  PR[91,3] = PR[90,3] + 11.289;
   1:L PR[91] R[100]mm/sec CNT100;
   1:  PR[91,1] = PR[90,1] + 1.252;
   1:  PR[91,2] = PR[90,2] + 3.696;
   1:  PR[91,3] = PR[90,3] + 11.292;
   1:L PR[91] R[100]mm/sec CNT100;
   1:  PR[91,1] = PR[90,1] + 0.910;
   1:  PR[91,2] = PR[90,2] + 3.517;
   1:  PR[91,3] = PR[90,3] + 11.295;
   1:L PR[91] R[100]mm/sec CNT100;
   1:  PR[91,1] = PR[90,1] + 0.499;
   1:  PR[91,2] = PR[90,2] + 3.376;
   1:  PR[91,3] = PR[90,3] + 11.297;
   1:L PR[91] R[100]mm/sec CNT100;
   1:  PR[91,1] = PR[90,1] + 0.087;
   1:  PR[91,2] = PR[90,2] + 3.307;
   1:  PR[91,3] = PR[90,3] + 11.300;
   1:L PR[91] R[100]mm/sec CNT100;
   1:  PR[91,1] = PR[90,1] + -0.331;
   1:  PR[91,3] = PR[90,3] + 11.302;
   1:L PR[91] R[100]mm/sec CNT100;
   1:  PR[91,1] = PR[90,1] + -0.746;
   1:  PR[91,2] = PR[90,2] + 3.378;
   1:  PR[91,3] = PR[90,3] + 11.305;
   1:L PR[91] R[100]mm/sec CNT100;
   1:  PR[91,1] = PR[90,1] + -1.128;
   1:  PR[91,2] = PR[90,2] + 3.507;
   1:  PR[91,3] = PR[90,3] + 11.308;
   1:L PR[91] R[100]mm/sec CNT100;
   1:  PR[91,1] = PR[90,1] + -1.497;
   1:  PR[91,2] = PR[90,2] + 3.698;
   1:  PR[91,3] = PR[90,3] + 11.310;
   1:L PR[91] R[100]mm/sec CNT100;
   1:  PR[91,1] = PR[90,1] + -1.899;
   1:  PR[91,2] = PR[90,2] + 3.996;
   1:  PR[91,3] = PR[90,3] + 11.313;
   1:L PR[91] R[100]mm/sec CNT100;
   1:  PR[91,1] = PR[90,1] + -2.131;
   1:  PR[91,2] = PR[90,2] + 4.220;
   1:  PR[91,3] = PR[90,3] + 11.316;
   1:L PR[91] R[100]mm/sec CNT100;
   1:  PR[91,1] = PR[90,1] + -2.395;
   1:  PR[91,2] = PR[90,2] + 4.536;
   1:  PR[91,3] = PR[90,3] + 11.318;
   1:L PR[91] R[100]mm/sec CNT100;
   1:  PR[91,1] = PR[90,1] + -2.627;
   1:  PR[91,2] = PR[90,2] + 4.887;
   1:  PR[91,3] = PR[90,3] + 11.321;
   1:L PR[91] R[100]mm/sec CNT100;
   1:  PR[91,1] = PR[90,1] + -2.824;
   1:  PR[91,2] = PR[90,2] + 5.271;
   1:  PR[91,3] = PR[90,3] + 11.323;
   1:L PR[91] R[100]mm/sec CNT100;
   1:  PR[91,1] = PR[90,1] + -3.191;
   1:  PR[91,2] = PR[90,2] + 6.264;
   1:  PR[91,3] = PR[90,3] + 11.326;
   1:L PR[91] R[100]mm/sec CNT100;
   1:  PR[91,1] = PR[90,1] + -3.514;
   1:  PR[91,2] = PR[90,2] + 7.053;
   1:  PR[91,3] = PR[90,3] + 11.333;
   1:L PR[91] R[100]mm/sec CNT100;
   1:  PR[91,1] = PR[90,1] + -3.875;
   1:  PR[91,2] = PR[90,2] + 7.826;
   1:  PR[91,3] = PR[90,3] + 11.338;
   1:L PR[91] R[100]mm/sec CNT100;
   1:  PR[91,1] = PR[90,1] + -4.277;
   1:  PR[91,2] = PR[90,2] + 8.584;
   1:  PR[91,3] = PR[90,3] + 11.344;
   1:L PR[91] R[100]mm/sec CNT100;
   1:  PR[91,1] = PR[90,1] + -4.715;
   1:  PR[91,2] = PR[90,2] + 9.322;
   1:  PR[91,3] = PR[90,3] + 11.349;
   1:L PR[91] R[100]mm/sec CNT100;
   1:  PR[91,1] = PR[90,1] + -5.189;
   1:  PR[91,2] = PR[90,2] + 10.038;
   1:  PR[91,3] = PR[90,3] + 11.354;
   1:L PR[91] R[100]mm/sec CNT100;
   1:  PR[91,1] = PR[90,1] + -5.698;
   1:  PR[91,2] = PR[90,2] + 10.728;
   1:  PR[91,3] = PR[90,3] + 11.360;
   1:L PR[91] R[100]mm/sec CNT100;
   1:  PR[91,1] = PR[90,1] + -6.242;
   1:  PR[91,2] = PR[90,2] + 11.391;
   1:  PR[91,3] = PR[90,3] + 11.365;
   1:L PR[91] R[100]mm/sec CNT100;
   1:  PR[91,1] = PR[90,1] + -6.819;
   1:  PR[91,2] = PR[90,2] + 12.026;
   1:  PR[91,3] = PR[90,3] + 11.371;
   1:L PR[91] R[100]mm/sec CNT100;
   1:  PR[91,1] = PR[90,1] + -7.193;
   1:  PR[91,2] = PR[90,2] + 12.401;
   1:  PR[91,3] = PR[90,3] + 11.376;
   1:L PR[91] R[100]mm/sec CNT100;
   1:  PR[91,1] = PR[90,1] + -7.425;
   1:  PR[91,2] = PR[90,2] + 12.629;
   1:  PR[91,3] = PR[90,3] + 11.380;
   1:L PR[91] R[100]mm/sec CNT100;
   1:  PR[91,1] = PR[90,1] + -8.063;
   1:  PR[91,2] = PR[90,2] + 13.204;
   1:  PR[91,3] = PR[90,3] + 11.382;
   1:L PR[91] R[100]mm/sec CNT100;
   1:  PR[91,1] = PR[90,1] + -8.730;
   1:  PR[91,2] = PR[90,2] + 13.747;
   1:  PR[91,3] = PR[90,3] + 11.387;
   1:L PR[91] R[100]mm/sec CNT100;
   1:  PR[91,1] = PR[90,1] + -8.985;
   1:  PR[91,2] = PR[90,2] + 13.936;
   1:  PR[91,3] = PR[90,3] + 11.393;
   1:L PR[91] R[100]mm/sec CNT100;
   1:  PR[91,1] = PR[90,1] + -9.420;
   1:  PR[91,2] = PR[90,2] + 14.254;
   1:  PR[91,3] = PR[90,3] + 11.395;
   1:L PR[91] R[100]mm/sec CNT100;
   1:  PR[91,1] = PR[90,1] + -10.136;
   1:  PR[91,2] = PR[90,2] + 14.728;
   1:  PR[91,3] = PR[90,3] + 11.398;
   1:L PR[91] R[100]mm/sec CNT100;
   1:  PR[91,1] = PR[90,1] + -10.874;
   1:  PR[91,2] = PR[90,2] + 15.166;
   1:  PR[91,3] = PR[90,3] + 11.403;
   1:L PR[91] R[100]mm/sec CNT100;
   1:  PR[91,1] = PR[90,1] + -11.633;
   1:  PR[91,2] = PR[90,2] + 15.568;
   1:  PR[91,3] = PR[90,3] + 11.409;
   1:L PR[91] R[100]mm/sec CNT100;
   1:  PR[91,1] = PR[90,1] + -12.420;
   1:  PR[91,2] = PR[90,2] + 15.937;
   1:  PR[91,3] = PR[90,3] + 11.414;
   1:L PR[91] R[100]mm/sec CNT100;
   1:  PR[91,1] = PR[90,1] + -13.133;
   1:  PR[91,2] = PR[90,2] + 16.233;
   1:  PR[91,3] = PR[90,3] + 11.420;
   1:L PR[91] R[100]mm/sec CNT100;
   1:  PR[91,1] = PR[90,1] + -13.894;
   1:  PR[91,2] = PR[90,2] + 16.508;
   1:  PR[91,3] = PR[90,3] + 11.425;
   1:L PR[91] R[100]mm/sec CNT100;
   1:  PR[91,1] = PR[90,1] + -14.667;
   1:  PR[91,2] = PR[90,2] + 16.749;
   1:  PR[91,3] = PR[90,3] + 11.430;
   1:L PR[91] R[100]mm/sec CNT100;
   1:  PR[91,1] = PR[90,1] + -15.453;
   1:  PR[91,2] = PR[90,2] + 16.954;
   1:  PR[91,3] = PR[90,3] + 11.435;
   1:L PR[91] R[100]mm/sec CNT100;
   1:  PR[91,1] = PR[90,1] + -16.250;
   1:  PR[91,2] = PR[90,2] + 17.123;
   1:  PR[91,3] = PR[90,3] + 11.440;
   1:L PR[91] R[100]mm/sec CNT100;
   1:  PR[91,1] = PR[90,1] + -17.055;
   1:  PR[91,2] = PR[90,2] + 17.255;
   1:  PR[91,3] = PR[90,3] + 11.445;
   1:L PR[91] R[100]mm/sec CNT100;
   1:  PR[91,1] = PR[90,1] + -17.868;
   1:  PR[91,2] = PR[90,2] + 17.350;
   1:  PR[91,3] = PR[90,3] + 11.450;
   1:L PR[91] R[100]mm/sec CNT100;
   1:  PR[91,1] = PR[90,1] + -18.686;
   1:  PR[91,2] = PR[90,2] + 17.407;
   1:  PR[91,3] = PR[90,3] + 11.456;
   1:L PR[91] R[100]mm/sec CNT100;
   1:  PR[91,1] = PR[90,1] + -19.508;
   1:  PR[91,2] = PR[90,2] + 17.426;
   1:  PR[91,3] = PR[90,3] + 11.461;
   1:L PR[91] R[100]mm/sec CNT100;
   1:  PR[91,1] = PR[90,1] + -20.332;
   1:  PR[91,2] = PR[90,2] + 17.406;
   1:  PR[91,3] = PR[90,3] + 11.466;
   1:L PR[91] R[100]mm/sec CNT100;
   1:  PR[91,1] = PR[90,1] + -21.156;
   1:  PR[91,2] = PR[90,2] + 17.348;
   1:  PR[91,3] = PR[90,3] + 11.471;
   1:L PR[91] R[100]mm/sec CNT100;
   1:  PR[91,1] = PR[90,1] + -21.977;
   1:  PR[91,2] = PR[90,2] + 17.250;
   1:  PR[91,3] = PR[90,3] + 11.476;
   1:L PR[91] R[100]mm/sec CNT100;
   1:  PR[91,1] = PR[90,1] + -22.817;
   1:  PR[91,2] = PR[90,2] + 17.109;
   1:  PR[91,3] = PR[90,3] + 11.482;
   1:L PR[91] R[100]mm/sec CNT100;
   1:  PR[91,1] = PR[90,1] + -23.651;
   1:  PR[91,2] = PR[90,2] + 16.927;
   1:  PR[91,3] = PR[90,3] + 11.487;
   1:L PR[91] R[100]mm/sec CNT100;
   1:  PR[91,1] = PR[90,1] + -24.474;
   1:  PR[91,2] = PR[90,2] + 16.704;
   1:  PR[91,3] = PR[90,3] + 11.492;
   1:L PR[91] R[100]mm/sec CNT100;
   1:  PR[91,1] = PR[90,1] + -25.284;
   1:  PR[91,2] = PR[90,2] + 16.441;
   1:  PR[91,3] = PR[90,3] + 11.498;
   1:L PR[91] R[100]mm/sec CNT100;
   1:  PR[91,1] = PR[90,1] + -26.079;
   1:  PR[91,2] = PR[90,2] + 16.139;
   1:  PR[91,3] = PR[90,3] + 11.503;
   1:L PR[91] R[100]mm/sec CNT100;
   1:  PR[91,1] = PR[90,1] + -26.857;
   1:  PR[91,2] = PR[90,2] + 15.799;
   1:  PR[91,3] = PR[90,3] + 11.509;
   1:L PR[91] R[100]mm/sec CNT100;
   1:  PR[91,1] = PR[90,1] + -27.616;
   1:  PR[91,2] = PR[90,2] + 15.422;
   1:  PR[91,3] = PR[90,3] + 11.514;
   1:L PR[91] R[100]mm/sec CNT100;
   1:  PR[91,1] = PR[90,1] + -28.355;
   1:  PR[91,2] = PR[90,2] + 15.009;
   1:  PR[91,3] = PR[90,3] + 11.519;
   1:L PR[91] R[100]mm/sec CNT100;
   1:  PR[91,1] = PR[90,1] + -29.072;
   1:  PR[91,2] = PR[90,2] + 14.560;
   1:  PR[91,3] = PR[90,3] + 11.525;
   1:L PR[91] R[100]mm/sec CNT100;
   1:  PR[91,1] = PR[90,1] + -29.765;
   1:  PR[91,2] = PR[90,2] + 14.078;
   1:  PR[91,3] = PR[90,3] + 11.530;
   1:L PR[91] R[100]mm/sec CNT100;
   1:  PR[91,1] = PR[90,1] + -30.432;
   1:  PR[91,2] = PR[90,2] + 13.563;
   1:  PR[91,3] = PR[90,3] + 11.535;
   1:L PR[91] R[100]mm/sec CNT100;
   1:  PR[91,1] = PR[90,1] + -31.073;
   1:  PR[91,2] = PR[90,2] + 13.017;
   1:  PR[91,3] = PR[90,3] + 11.541;
   1:L PR[91] R[100]mm/sec CNT100;
   1:  PR[91,1] = PR[90,1] + -31.685;
   1:  PR[91,2] = PR[90,2] + 12.440;
   1:  PR[91,3] = PR[90,3] + 11.546;
   1:L PR[91] R[100]mm/sec CNT100;
   1:  PR[91,1] = PR[90,1] + -32.267;
   1:  PR[91,2] = PR[90,2] + 11.834;
   1:  PR[91,3] = PR[90,3] + 11.552;
   1:L PR[91] R[100]mm/sec CNT100;
   1:  PR[91,1] = PR[90,1] + -32.818;
   1:  PR[91,2] = PR[90,2] + 11.201;
   1:  PR[91,3] = PR[90,3] + 11.557;
   1:L PR[91] R[100]mm/sec CNT100;
   1:  PR[91,1] = PR[90,1] + -33.336;
   1:  PR[91,2] = PR[90,2] + 10.542;
   1:  PR[91,3] = PR[90,3] + 11.562;
   1:L PR[91] R[100]mm/sec CNT100;
   1:  PR[91,1] = PR[90,1] + -33.821;
   1:  PR[91,2] = PR[90,2] + 9.858;
   1:  PR[91,3] = PR[90,3] + 11.567;
   1:L PR[91] R[100]mm/sec CNT100;
   1:  PR[91,1] = PR[90,1] + -34.272;
   1:  PR[91,2] = PR[90,2] + 9.151;
   1:  PR[91,3] = PR[90,3] + 11.573;
   1:L PR[91] R[100]mm/sec CNT100;
   1:  PR[91,1] = PR[90,1] + -34.687;
   1:  PR[91,2] = PR[90,2] + 8.423;
   1:  PR[91,3] = PR[90,3] + 11.578;
   1:L PR[91] R[100]mm/sec CNT100;
   1:  PR[91,1] = PR[90,1] + -35.065;
   1:  PR[91,2] = PR[90,2] + 7.677;
   1:  PR[91,3] = PR[90,3] + 11.583;
   1:L PR[91] R[100]mm/sec CNT100;
   1:  PR[91,1] = PR[90,1] + -35.406;
   1:  PR[91,2] = PR[90,2] + 6.915;
   1:  PR[91,3] = PR[90,3] + 11.589;
   1:L PR[91] R[100]mm/sec CNT100;
   1:  PR[91,1] = PR[90,1] + -35.714;
   1:  PR[91,2] = PR[90,2] + 6.122;
   1:  PR[91,3] = PR[90,3] + 11.594;
   1:L PR[91] R[100]mm/sec CNT100;
   1:  PR[91,1] = PR[90,1] + -35.973;
   1:  PR[91,2] = PR[90,2] + 5.348;
   1:  PR[91,3] = PR[90,3] + 11.599;
   1:L PR[91] R[100]mm/sec CNT100;
   1:  PR[91,1] = PR[90,1] + -36.196;
   1:  PR[91,2] = PR[90,2] + 4.551;
   1:  PR[91,3] = PR[90,3] + 11.605;
   1:L PR[91] R[100]mm/sec CNT100;
   1:  PR[91,1] = PR[90,1] + -36.381;
   1:  PR[91,2] = PR[90,2] + 3.736;
   1:  PR[91,3] = PR[90,3] + 11.610;
   1:L PR[91] R[100]mm/sec CNT100;
   1:  PR[91,1] = PR[90,1] + -36.522;
   1:  PR[91,2] = PR[90,2] + 2.935;
   1:  PR[91,3] = PR[90,3] + 11.615;
   1:L PR[91] R[100]mm/sec CNT100;
   1:  PR[91,1] = PR[90,1] + -36.624;
   1:  PR[91,2] = PR[90,2] + 2.109;
   1:  PR[91,3] = PR[90,3] + 11.620;
   1:L PR[91] R[100]mm/sec CNT100;
   1:  PR[91,1] = PR[90,1] + -36.686;
   1:  PR[91,2] = PR[90,2] + 1.273;
   1:  PR[91,3] = PR[90,3] + 11.626;
   1:L PR[91] R[100]mm/sec CNT100;
   1:  PR[91,1] = PR[90,1] + -36.707;
   1:  PR[91,2] = PR[90,2] + 0.428;
   1:  PR[91,3] = PR[90,3] + 11.631;
   1:L PR[91] R[100]mm/sec CNT100;
   1:  PR[91,1] = PR[90,1] + -36.686;
   1:  PR[91,2] = PR[90,2] + -0.418;
   1:  PR[91,3] = PR[90,3] + 11.636;
   1:L PR[91] R[100]mm/sec CNT100;
   1:  PR[91,1] = PR[90,1] + -36.624;
   1:  PR[91,2] = PR[90,2] + -1.254;
   1:  PR[91,3] = PR[90,3] + 11.642;
   1:L PR[91] R[100]mm/sec CNT100;
   1:  PR[91,1] = PR[90,1] + -36.522;
   1:  PR[91,2] = PR[90,2] + -2.080;
   1:  PR[91,3] = PR[90,3] + 11.647;
   1:L PR[91] R[100]mm/sec CNT100;
   1:  PR[91,1] = PR[90,1] + -36.379;
   1:  PR[91,2] = PR[90,2] + -2.895;
   1:  PR[91,3] = PR[90,3] + 11.652;
   1:L PR[91] R[100]mm/sec CNT100;
   1:  PR[91,1] = PR[90,1] + -36.195;
   1:  PR[91,2] = PR[90,2] + -3.701;
   1:  PR[91,3] = PR[90,3] + 11.657;
   1:L PR[91] R[100]mm/sec CNT100;
   1:  PR[91,1] = PR[90,1] + -35.972;
   1:  PR[91,2] = PR[90,2] + -4.498;
   1:  PR[91,3] = PR[90,3] + 11.663;
   1:L PR[91] R[100]mm/sec CNT100;
   1:  PR[91,1] = PR[90,1] + -35.708;
   1:  PR[91,2] = PR[90,2] + -5.284;
   1:  PR[91,3] = PR[90,3] + 11.668;
   1:L PR[91] R[100]mm/sec CNT100;
   1:  PR[91,1] = PR[90,1] + -35.406;
   1:  PR[91,2] = PR[90,2] + -6.060;
   1:  PR[91,3] = PR[90,3] + 11.673;
   1:L PR[91] R[100]mm/sec CNT100;
   1:  PR[91,1] = PR[90,1] + -35.065;
   1:  PR[91,2] = PR[90,2] + -6.822;
   1:  PR[91,3] = PR[90,3] + 11.678;
   1:L PR[91] R[100]mm/sec CNT100;
   1:  PR[91,1] = PR[90,1] + -34.687;
   1:  PR[91,2] = PR[90,2] + -7.568;
   1:  PR[91,3] = PR[90,3] + 11.684;
   1:L PR[91] R[100]mm/sec CNT100;
   1:  PR[91,1] = PR[90,1] + -34.272;
   1:  PR[91,2] = PR[90,2] + -8.296;
   1:  PR[91,3] = PR[90,3] + 11.689;
   1:L PR[91] R[100]mm/sec CNT100;
   1:  PR[91,1] = PR[90,1] + -33.821;
   1:  PR[91,2] = PR[90,2] + -9.003;
   1:  PR[91,3] = PR[90,3] + 11.694;
   1:L PR[91] R[100]mm/sec CNT100;
   1:  PR[91,1] = PR[90,1] + -33.336;
   1:  PR[91,2] = PR[90,2] + -9.687;
   1:  PR[91,3] = PR[90,3] + 11.700;
   1:L PR[91] R[100]mm/sec CNT100;
   1:  PR[91,1] = PR[90,1] + -32.818;
   1:  PR[91,2] = PR[90,2] + -10.346;
   1:  PR[91,3] = PR[90,3] + 11.705;
   1:L PR[91] R[100]mm/sec CNT100;
   1:  PR[91,1] = PR[90,1] + -32.267;
   1:  PR[91,2] = PR[90,2] + -10.979;
   1:  PR[91,3] = PR[90,3] + 11.710;
   1:L PR[91] R[100]mm/sec CNT100;
   1:  PR[91,1] = PR[90,1] + -31.684;
   1:  PR[91,2] = PR[90,2] + -11.585;
   1:  PR[91,3] = PR[90,3] + 11.716;
   1:L PR[91] R[100]mm/sec CNT100;
   1:  PR[91,1] = PR[90,1] + -31.073;
   1:  PR[91,2] = PR[90,2] + -12.161;
   1:  PR[91,3] = PR[90,3] + 11.721;
   1:L PR[91] R[100]mm/sec CNT100;
   1:  PR[91,1] = PR[90,1] + -30.432;
   1:  PR[91,2] = PR[90,2] + -12.708;
   1:  PR[91,3] = PR[90,3] + 11.726;
   1:L PR[91] R[100]mm/sec CNT100;
   1:  PR[91,1] = PR[90,1] + -29.765;
   1:  PR[91,2] = PR[90,2] + -13.223;
   1:  PR[91,3] = PR[90,3] + 11.732;
   1:L PR[91] R[100]mm/sec CNT100;
   1:  PR[91,1] = PR[90,1] + -29.072;
   1:  PR[91,2] = PR[90,2] + -13.705;
   1:  PR[91,3] = PR[90,3] + 11.737;
   1:L PR[91] R[100]mm/sec CNT100;
   1:  PR[91,1] = PR[90,1] + -28.355;
   1:  PR[91,2] = PR[90,2] + -14.153;
   1:  PR[91,3] = PR[90,3] + 11.742;
   1:L PR[91] R[100]mm/sec CNT100;
   1:  PR[91,1] = PR[90,1] + -27.616;
   1:  PR[91,2] = PR[90,2] + -14.567;
   1:  PR[91,3] = PR[90,3] + 11.748;
   1:L PR[91] R[100]mm/sec CNT100;
   1:  PR[91,1] = PR[90,1] + -26.857;
   1:  PR[91,2] = PR[90,2] + -14.944;
   1:  PR[91,3] = PR[90,3] + 11.753;
   1:L PR[91] R[100]mm/sec CNT100;
   1:  PR[91,1] = PR[90,1] + -26.079;
   1:  PR[91,2] = PR[90,2] + -15.284;
   1:  PR[91,3] = PR[90,3] + 11.758;
   1:L PR[91] R[100]mm/sec CNT100;
   1:  PR[91,1] = PR[90,1] + -25.284;
   1:  PR[91,2] = PR[90,2] + -15.586;
   1:  PR[91,3] = PR[90,3] + 11.764;
   1:L PR[91] R[100]mm/sec CNT100;
   1:  PR[91,1] = PR[90,1] + -24.474;
   1:  PR[91,2] = PR[90,2] + -15.849;
   1:  PR[91,3] = PR[90,3] + 11.769;
   1:L PR[91] R[100]mm/sec CNT100;
   1:  PR[91,1] = PR[90,1] + -23.651;
   1:  PR[91,2] = PR[90,2] + -16.071;
   1:  PR[91,3] = PR[90,3] + 11.774;
   1:L PR[91] R[100]mm/sec CNT100;
   1:  PR[91,1] = PR[90,1] + -22.817;
   1:  PR[91,2] = PR[90,2] + -16.254;
   1:  PR[91,3] = PR[90,3] + 11.780;
   1:L PR[91] R[100]mm/sec CNT100;
   1:  PR[91,1] = PR[90,1] + -21.969;
   1:  PR[91,2] = PR[90,2] + -16.396;
   1:  PR[91,3] = PR[90,3] + 11.785;
   1:L PR[91] R[100]mm/sec CNT100;
   1:  PR[91,1] = PR[90,1] + -21.157;
   1:  PR[91,2] = PR[90,2] + -16.492;
   1:  PR[91,3] = PR[90,3] + 11.791;
   1:L PR[91] R[100]mm/sec CNT100;
   1:  PR[91,1] = PR[90,1] + -20.193;
   1:  PR[91,2] = PR[90,2] + -16.557;
   1:  PR[91,3] = PR[90,3] + 11.796;
   1:L PR[91] R[100]mm/sec CNT100;
   1:  PR[91,1] = PR[90,1] + -19.509;
   1:  PR[91,2] = PR[90,2] + -16.571;
   1:  PR[91,3] = PR[90,3] + 11.802;
   1:L PR[91] R[100]mm/sec CNT100;
   1:  PR[91,1] = PR[90,1] + -18.689;
   1:  PR[91,2] = PR[90,2] + -16.552;
   1:  PR[91,3] = PR[90,3] + 11.806;
   1:L PR[91] R[100]mm/sec CNT100;
   1:  PR[91,1] = PR[90,1] + -17.523;
   1:  PR[91,2] = PR[90,2] + -16.459;
   1:  PR[91,3] = PR[90,3] + 11.812;
   1:L PR[91] R[100]mm/sec CNT100;
   1:  PR[91,1] = PR[90,1] + -17.058;
   1:  PR[91,2] = PR[90,2] + -16.400;
   1:  PR[91,3] = PR[90,3] + 11.819;
   1:L PR[91] R[100]mm/sec CNT100;
   1:  PR[91,1] = PR[90,1] + -16.250;
   1:  PR[91,2] = PR[90,2] + -16.268;
   1:  PR[91,3] = PR[90,3] + 11.822;
   1:L PR[91] R[100]mm/sec CNT100;
   1:  PR[91,1] = PR[90,1] + -15.451;
   1:  PR[91,2] = PR[90,2] + -16.098;
   1:  PR[91,3] = PR[90,3] + 11.827;
   1:L PR[91] R[100]mm/sec CNT100;
   1:  PR[91,1] = PR[90,1] + -14.920;
   1:  PR[91,2] = PR[90,2] + -15.964;
   1:  PR[91,3] = PR[90,3] + 11.832;
   1:L PR[91] R[100]mm/sec CNT100;
   1:  PR[91,1] = PR[90,1] + -13.892;
   1:  PR[91,2] = PR[90,2] + -15.652;
   1:  PR[91,3] = PR[90,3] + 11.836;
   1:L PR[91] R[100]mm/sec CNT100;
   1:  PR[91,1] = PR[90,1] + -13.134;
   1:  PR[91,2] = PR[90,2] + -15.378;
   1:  PR[91,3] = PR[90,3] + 11.843;
   1:L PR[91] R[100]mm/sec CNT100;
   1:  PR[91,1] = PR[90,1] + -12.389;
   1:  PR[91,2] = PR[90,2] + -15.069;
   1:  PR[91,3] = PR[90,3] + 11.848;
   1:L PR[91] R[100]mm/sec CNT100;
   1:  PR[91,1] = PR[90,1] + -11.633;
   1:  PR[91,2] = PR[90,2] + -14.713;
   1:  PR[91,3] = PR[90,3] + 11.853;
   1:L PR[91] R[100]mm/sec CNT100;
   1:  PR[91,1] = PR[90,1] + -10.875;
   1:  PR[91,2] = PR[90,2] + -14.311;
   1:  PR[91,3] = PR[90,3] + 11.858;
   1:L PR[91] R[100]mm/sec CNT100;
   1:  PR[91,1] = PR[90,1] + -10.136;
   1:  PR[91,2] = PR[90,2] + -13.873;
   1:  PR[91,3] = PR[90,3] + 11.864;
   1:L PR[91] R[100]mm/sec CNT100;
   1:  PR[91,1] = PR[90,1] + -9.635;
   1:  PR[91,2] = PR[90,2] + -13.543;
   1:  PR[91,3] = PR[90,3] + 11.869;
   1:L PR[91] R[100]mm/sec CNT100;
   1:  PR[91,1] = PR[90,1] + -8.727;
   1:  PR[91,2] = PR[90,2] + -12.889;
   1:  PR[91,3] = PR[90,3] + 11.873;
   1:L PR[91] R[100]mm/sec CNT100;
   1:  PR[91,1] = PR[90,1] + -8.063;
   1:  PR[91,2] = PR[90,2] + -12.349;
   1:  PR[91,3] = PR[90,3] + 11.880;
   1:L PR[91] R[100]mm/sec CNT100;
   1:  PR[91,1] = PR[90,1] + -7.425;
   1:  PR[91,2] = PR[90,2] + -11.774;
   1:  PR[91,3] = PR[90,3] + 11.885;
   1:L PR[91] R[100]mm/sec CNT100;
   1:  PR[91,1] = PR[90,1] + -7.193;
   1:  PR[91,2] = PR[90,2] + -11.546;
   1:  PR[91,3] = PR[90,3] + 11.891;
   1:L PR[91] R[100]mm/sec CNT100;
   1:  PR[91,1] = PR[90,1] + -6.819;
   1:  PR[91,2] = PR[90,2] + -11.171;
   1:  PR[91,3] = PR[90,3] + 11.893;
   1:L PR[91] R[100]mm/sec CNT100;
   1:  PR[91,1] = PR[90,1] + -6.243;
   1:  PR[91,2] = PR[90,2] + -10.537;
   1:  PR[91,3] = PR[90,3] + 11.896;
   1:L PR[91] R[100]mm/sec CNT100;
   1:  PR[91,1] = PR[90,1] + -5.613;
   1:  PR[91,2] = PR[90,2] + -9.759;
   1:  PR[91,3] = PR[90,3] + 11.902;
   1:L PR[91] R[100]mm/sec CNT100;
   1:  PR[91,1] = PR[90,1] + -5.189;
   1:  PR[91,2] = PR[90,2] + -9.183;
   1:  PR[91,3] = PR[90,3] + 11.908;
   1:L PR[91] R[100]mm/sec CNT100;
   1:  PR[91,1] = PR[90,1] + -4.702;
   1:  PR[91,2] = PR[90,2] + -8.446;
   1:  PR[91,3] = PR[90,3] + 11.912;
   1:L PR[91] R[100]mm/sec CNT100;
   1:  PR[91,1] = PR[90,1] + -4.277;
   1:  PR[91,2] = PR[90,2] + -7.729;
   1:  PR[91,3] = PR[90,3] + 11.918;
   1:L PR[91] R[100]mm/sec CNT100;
   1:  PR[91,1] = PR[90,1] + -3.876;
   1:  PR[91,2] = PR[90,2] + -6.971;
   1:  PR[91,3] = PR[90,3] + 11.923;
   1:L PR[91] R[100]mm/sec CNT100;
   1:  PR[91,1] = PR[90,1] + -3.514;
   1:  PR[91,2] = PR[90,2] + -6.198;
   1:  PR[91,3] = PR[90,3] + 11.929;
   1:L PR[91] R[100]mm/sec CNT100;
   1:  PR[91,1] = PR[90,1] + -3.191;
   1:  PR[91,2] = PR[90,2] + -5.409;
   1:  PR[91,3] = PR[90,3] + 11.934;
   1:L PR[91] R[100]mm/sec CNT100;
   1:  PR[91,1] = PR[90,1] + -2.824;
   1:  PR[91,2] = PR[90,2] + -4.415;
   1:  PR[91,3] = PR[90,3] + 11.940;
   1:L PR[91] R[100]mm/sec CNT100;
   1:  PR[91,1] = PR[90,1] + -2.626;
   1:  PR[91,2] = PR[90,2] + -4.031;
   1:  PR[91,3] = PR[90,3] + 11.946;
   1:L PR[91] R[100]mm/sec CNT100;
   1:  PR[91,1] = PR[90,1] + -2.395;
   1:  PR[91,2] = PR[90,2] + -3.679;
   1:  PR[91,3] = PR[90,3] + 11.949;
   1:L PR[91] R[100]mm/sec CNT100;
   1:  PR[91,1] = PR[90,1] + -2.127;
   1:  PR[91,2] = PR[90,2] + -3.360;
   1:  PR[91,3] = PR[90,3] + 11.952;
   1:L PR[91] R[100]mm/sec CNT100;
   1:  PR[91,1] = PR[90,1] + -1.825;
   1:  PR[91,2] = PR[90,2] + -3.078;
   1:  PR[91,3] = PR[90,3] + 11.954;
   1:L PR[91] R[100]mm/sec CNT100;
   1:  PR[91,1] = PR[90,1] + -1.492;
   1:  PR[91,2] = PR[90,2] + -2.841;
   1:  PR[91,3] = PR[90,3] + 11.957;
   1:L PR[91] R[100]mm/sec CNT100;
   1:  PR[91,1] = PR[90,1] + -1.153;
   1:  PR[91,2] = PR[90,2] + -2.663;
   1:  PR[91,3] = PR[90,3] + 11.960;
   1:L PR[91] R[100]mm/sec CNT100;
   1:  PR[91,1] = PR[90,1] + -0.739;
   1:  PR[91,2] = PR[90,2] + -2.520;
   1:  PR[91,3] = PR[90,3] + 11.962;
   1:L PR[91] R[100]mm/sec CNT100;
   1:  PR[91,1] = PR[90,1] + -0.329;
   1:  PR[91,2] = PR[90,2] + -2.452;
   1:  PR[91,3] = PR[90,3] + 11.965;
   1:L PR[91] R[100]mm/sec CNT100;
   1:  PR[91,1] = PR[90,1] + 0.089;
   1:  PR[91,3] = PR[90,3] + 11.967;
   1:L PR[91] R[100]mm/sec CNT100;
   1:  PR[91] = PR[90];
   1:  PR[91,1] = PR[90,1] + 0.253;
   1:  PR[91,2] = PR[90,2] + -3.587;
   1:  PR[91,3] = PR[90,3] + 13.300;
   1:L PR[91] R[100]mm/sec CNT100;
   1:  PR[91,1] = PR[90,1] + 0.757;
   1:  PR[91,2] = PR[90,2] + -3.715;
   1:  PR[91,3] = PR[90,3] + 11.972;
   1:L PR[91] R[100]mm/sec CNT100;
   1:  PR[91,1] = PR[90,1] + 1.032;
   1:  PR[91,2] = PR[90,2] + -3.832;
   1:  PR[91,3] = PR[90,3] + 11.975;
   1:L PR[91] R[100]mm/sec CNT100;
   1:  PR[91,1] = PR[90,1] + 1.382;
   1:  PR[91,2] = PR[90,2] + -4.035;
   1:  PR[91,3] = PR[90,3] + 11.977;
   1:L PR[91] R[100]mm/sec CNT100;
   1:  PR[91,1] = PR[90,1] + 1.703;
   1:  PR[91,2] = PR[90,2] + -4.286;
   1:  PR[91,3] = PR[90,3] + 11.980;
   1:L PR[91] R[100]mm/sec CNT100;
   1:  PR[91,1] = PR[90,1] + 1.896;
   1:  PR[91,2] = PR[90,2] + -4.475;
   1:  PR[91,3] = PR[90,3] + 11.983;
   1:L PR[91] R[100]mm/sec CNT100;
   1:  PR[91,1] = PR[90,1] + 2.196;
   1:  PR[91,2] = PR[90,2] + -4.835;
   1:  PR[91,3] = PR[90,3] + 11.984;
   1:L PR[91] R[100]mm/sec CNT100;
   1:  PR[91,1] = PR[90,1] + 2.477;
   1:  PR[91,2] = PR[90,2] + -5.287;
   1:  PR[91,3] = PR[90,3] + 11.987;
   1:L PR[91] R[100]mm/sec CNT100;
   1:  PR[91,1] = PR[90,1] + 3.101;
   1:  PR[91,2] = PR[90,2] + -6.687;
   1:  PR[91,3] = PR[90,3] + 11.991;
   1:L PR[91] R[100]mm/sec CNT100;
   1:  PR[91,1] = PR[90,1] + 3.332;
   1:  PR[91,2] = PR[90,2] + -7.144;
   1:  PR[91,3] = PR[90,3] + 12.001;
   1:L PR[91] R[100]mm/sec CNT100;
   1:  PR[91,1] = PR[90,1] + 3.494;
   1:  PR[91,2] = PR[90,2] + -7.455;
   1:  PR[91,3] = PR[90,3] + 12.004;
   1:L PR[91] R[100]mm/sec CNT100;
   1:  PR[91,1] = PR[90,1] + 3.930;
   1:  PR[91,2] = PR[90,2] + -8.213;
   1:  PR[91,3] = PR[90,3] + 12.006;
   1:L PR[91] R[100]mm/sec CNT100;
   1:  PR[91,1] = PR[90,1] + 4.403;
   1:  PR[91,2] = PR[90,2] + -8.949;
   1:  PR[91,3] = PR[90,3] + 12.012;
   1:L PR[91] R[100]mm/sec CNT100;
   1:  PR[91,1] = PR[90,1] + 4.914;
   1:  PR[91,2] = PR[90,2] + -9.662;
   1:  PR[91,3] = PR[90,3] + 12.018;
   1:L PR[91] R[100]mm/sec CNT100;
   1:  PR[91,1] = PR[90,1] + 5.461;
   1:  PR[91,2] = PR[90,2] + -10.348;
   1:  PR[91,3] = PR[90,3] + 12.023;
   1:L PR[91] R[100]mm/sec CNT100;
   1:  PR[91,1] = PR[90,1] + 6.042;
   1:  PR[91,2] = PR[90,2] + -11.004;
   1:  PR[91,3] = PR[90,3] + 12.029;
   1:L PR[91] R[100]mm/sec CNT100;
   1:  PR[91,1] = PR[90,1] + 6.669;
   1:  PR[91,2] = PR[90,2] + -11.642;
   1:  PR[91,3] = PR[90,3] + 12.034;
   1:L PR[91] R[100]mm/sec CNT100;
   1:  PR[91,1] = PR[90,1] + 7.300;
   1:  PR[91,2] = PR[90,2] + -12.223;
   1:  PR[91,3] = PR[90,3] + 12.040;
   1:L PR[91] R[100]mm/sec CNT100;
   1:  PR[91,1] = PR[90,1] + 7.972;
   1:  PR[91,2] = PR[90,2] + -12.782;
   1:  PR[91,3] = PR[90,3] + 12.046;
   1:L PR[91] R[100]mm/sec CNT100;
   1:  PR[91,1] = PR[90,1] + 8.671;
   1:  PR[91,2] = PR[90,2] + -13.307;
   1:  PR[91,3] = PR[90,3] + 12.051;
   1:L PR[91] R[100]mm/sec CNT100;
   1:  PR[91,1] = PR[90,1] + 9.134;
   1:  PR[91,2] = PR[90,2] + -13.622;
   1:  PR[91,3] = PR[90,3] + 12.057;
   1:L PR[91] R[100]mm/sec CNT100;
   1:  PR[91,1] = PR[90,1] + 9.393;
   1:  PR[91,2] = PR[90,2] + -13.795;
   1:  PR[91,3] = PR[90,3] + 12.061;
   1:L PR[91] R[100]mm/sec CNT100;
   1:  PR[91,1] = PR[90,1] + 10.142;
   1:  PR[91,2] = PR[90,2] + -14.248;
   1:  PR[91,3] = PR[90,3] + 12.063;
   1:L PR[91] R[100]mm/sec CNT100;
   1:  PR[91,1] = PR[90,1] + 10.911;
   1:  PR[91,2] = PR[90,2] + -14.663;
   1:  PR[91,3] = PR[90,3] + 12.068;
   1:L PR[91] R[100]mm/sec CNT100;
   1:  PR[91,1] = PR[90,1] + 11.699;
   1:  PR[91,2] = PR[90,2] + -15.040;
   1:  PR[91,3] = PR[90,3] + 12.074;
   1:L PR[91] R[100]mm/sec CNT100;
   1:  PR[91,1] = PR[90,1] + 12.504;
   1:  PR[91,2] = PR[90,2] + -15.378;
   1:  PR[91,3] = PR[90,3] + 12.080;
   1:L PR[91] R[100]mm/sec CNT100;
   1:  PR[91,1] = PR[90,1] + 13.324;
   1:  PR[91,2] = PR[90,2] + -15.676;
   1:  PR[91,3] = PR[90,3] + 12.085;
   1:L PR[91] R[100]mm/sec CNT100;
   1:  PR[91,1] = PR[90,1] + 14.155;
   1:  PR[91,2] = PR[90,2] + -15.934;
   1:  PR[91,3] = PR[90,3] + 12.091;
   1:L PR[91] R[100]mm/sec CNT100;
   1:  PR[91,1] = PR[90,1] + 14.995;
   1:  PR[91,2] = PR[90,2] + -16.151;
   1:  PR[91,3] = PR[90,3] + 12.096;
   1:L PR[91] R[100]mm/sec CNT100;
   1:  PR[91,1] = PR[90,1] + 15.843;
   1:  PR[91,2] = PR[90,2] + -16.326;
   1:  PR[91,3] = PR[90,3] + 12.102;
   1:L PR[91] R[100]mm/sec CNT100;
   1:  PR[91,1] = PR[90,1] + 16.411;
   1:  PR[91,2] = PR[90,2] + -16.416;
   1:  PR[91,3] = PR[90,3] + 12.108;
   1:L PR[91] R[100]mm/sec CNT100;
   1:  PR[91,1] = PR[90,1] + 17.557;
   1:  PR[91,2] = PR[90,2] + -16.552;
   1:  PR[91,3] = PR[90,3] + 12.111;
   1:L PR[91] R[100]mm/sec CNT100;
   1:  PR[91,1] = PR[90,1] + 18.414;
   1:  PR[91,2] = PR[90,2] + -16.601;
   1:  PR[91,3] = PR[90,3] + 12.119;
   1:L PR[91] R[100]mm/sec CNT100;
   1:  PR[91,1] = PR[90,1] + 19.274;
   1:  PR[91,2] = PR[90,2] + -16.610;
   1:  PR[91,3] = PR[90,3] + 12.124;
   1:L PR[91] R[100]mm/sec CNT100;
   1:  PR[91,1] = PR[90,1] + 20.132;
   1:  PR[91,2] = PR[90,2] + -16.576;
   1:  PR[91,3] = PR[90,3] + 12.130;
   1:L PR[91] R[100]mm/sec CNT100;
   1:  PR[91,1] = PR[90,1] + 20.986;
   1:  PR[91,2] = PR[90,2] + -16.502;
   1:  PR[91,3] = PR[90,3] + 12.135;
   1:L PR[91] R[100]mm/sec CNT100;
   1:  PR[91,1] = PR[90,1] + 21.834;
   1:  PR[91,2] = PR[90,2] + -16.386;
   1:  PR[91,3] = PR[90,3] + 12.141;
   1:L PR[91] R[100]mm/sec CNT100;
   1:  PR[91,1] = PR[90,1] + 22.674;
   1:  PR[91,2] = PR[90,2] + -16.230;
   1:  PR[91,3] = PR[90,3] + 12.146;
   1:L PR[91] R[100]mm/sec CNT100;
   1:  PR[91,1] = PR[90,1] + 23.470;
   1:  PR[91,2] = PR[90,2] + -16.042;
   1:  PR[91,3] = PR[90,3] + 12.152;
   1:L PR[91] R[100]mm/sec CNT100;
   1:  PR[91,1] = PR[90,1] + 24.259;
   1:  PR[91,2] = PR[90,2] + -15.816;
   1:  PR[91,3] = PR[90,3] + 12.157;
   1:L PR[91] R[100]mm/sec CNT100;
   1:  PR[91,1] = PR[90,1] + 25.039;
   1:  PR[91,2] = PR[90,2] + -15.553;
   1:  PR[91,3] = PR[90,3] + 12.162;
   1:L PR[91] R[100]mm/sec CNT100;
   1:  PR[91,1] = PR[90,1] + 25.807;
   1:  PR[91,2] = PR[90,2] + -15.253;
   1:  PR[91,3] = PR[90,3] + 12.168;
   1:L PR[91] R[100]mm/sec CNT100;
   1:  PR[91,1] = PR[90,1] + 26.561;
   1:  PR[91,2] = PR[90,2] + -14.917;
   1:  PR[91,3] = PR[90,3] + 12.173;
   1:L PR[91] R[100]mm/sec CNT100;
   1:  PR[91,1] = PR[90,1] + 27.300;
   1:  PR[91,2] = PR[90,2] + -14.545;
   1:  PR[91,3] = PR[90,3] + 12.178;
   1:L PR[91] R[100]mm/sec CNT100;
   1:  PR[91,1] = PR[90,1] + 28.021;
   1:  PR[91,2] = PR[90,2] + -14.138;
   1:  PR[91,3] = PR[90,3] + 12.184;
   1:L PR[91] R[100]mm/sec CNT100;
   1:  PR[91,1] = PR[90,1] + 28.722;
   1:  PR[91,2] = PR[90,2] + -13.697;
   1:  PR[91,3] = PR[90,3] + 12.189;
   1:L PR[91] R[100]mm/sec CNT100;
   1:  PR[91,1] = PR[90,1] + 29.403;
   1:  PR[91,2] = PR[90,2] + -13.221;
   1:  PR[91,3] = PR[90,3] + 12.194;
   1:L PR[91] R[100]mm/sec CNT100;
   1:  PR[91,1] = PR[90,1] + 30.060;
   1:  PR[91,2] = PR[90,2] + -12.713;
   1:  PR[91,3] = PR[90,3] + 12.200;
   1:L PR[91] R[100]mm/sec CNT100;
   1:  PR[91,1] = PR[90,1] + 30.693;
   1:  PR[91,2] = PR[90,2] + -12.173;
   1:  PR[91,3] = PR[90,3] + 12.205;
   1:L PR[91] R[100]mm/sec CNT100;
   1:  PR[91,1] = PR[90,1] + 31.299;
   1:  PR[91,2] = PR[90,2] + -11.602;
   1:  PR[91,3] = PR[90,3] + 12.211;
   1:L PR[91] R[100]mm/sec CNT100;
   1:  PR[91,1] = PR[90,1] + 31.878;
   1:  PR[91,2] = PR[90,2] + -11.001;
   1:  PR[91,3] = PR[90,3] + 12.216;
   1:L PR[91] R[100]mm/sec CNT100;
   1:  PR[91,1] = PR[90,1] + 32.427;
   1:  PR[91,2] = PR[90,2] + -10.372;
   1:  PR[91,3] = PR[90,3] + 12.221;
   1:L PR[91] R[100]mm/sec CNT100;
   1:  PR[91,1] = PR[90,1] + 32.945;
   1:  PR[91,2] = PR[90,2] + -9.715;
   1:  PR[91,3] = PR[90,3] + 12.227;
   1:L PR[91] R[100]mm/sec CNT100;
   1:  PR[91,1] = PR[90,1] + 33.430;
   1:  PR[91,2] = PR[90,2] + -9.033;
   1:  PR[91,3] = PR[90,3] + 12.232;
   1:L PR[91] R[100]mm/sec CNT100;
   1:  PR[91,1] = PR[90,1] + 33.882;
   1:  PR[91,2] = PR[90,2] + -8.327;
   1:  PR[91,3] = PR[90,3] + 12.237;
   1:L PR[91] R[100]mm/sec CNT100;
   1:  PR[91,1] = PR[90,1] + 34.300;
   1:  PR[91,2] = PR[90,2] + -7.600;
   1:  PR[91,3] = PR[90,3] + 12.243;
   1:L PR[91] R[100]mm/sec CNT100;
   1:  PR[91,1] = PR[90,1] + 34.681;
   1:  PR[91,2] = PR[90,2] + -6.854;
   1:  PR[91,3] = PR[90,3] + 12.248;
   1:L PR[91] R[100]mm/sec CNT100;
   1:  PR[91,1] = PR[90,1] + 35.025;
   1:  PR[91,2] = PR[90,2] + -6.091;
   1:  PR[91,3] = PR[90,3] + 12.254;
   1:L PR[91] R[100]mm/sec CNT100;
   1:  PR[91,1] = PR[90,1] + 35.331;
   1:  PR[91,2] = PR[90,2] + -5.315;
   1:  PR[91,3] = PR[90,3] + 12.259;
   1:L PR[91] R[100]mm/sec CNT100;
   1:  PR[91,1] = PR[90,1] + 35.596;
   1:  PR[91,2] = PR[90,2] + -4.527;
   1:  PR[91,3] = PR[90,3] + 12.264;
   1:L PR[91] R[100]mm/sec CNT100;
   1:  PR[91,1] = PR[90,1] + 35.822;
   1:  PR[91,2] = PR[90,2] + -3.729;
   1:  PR[91,3] = PR[90,3] + 12.270;
   1:L PR[91] R[100]mm/sec CNT100;
   1:  PR[91,1] = PR[90,1] + 36.008;
   1:  PR[91,2] = PR[90,2] + -2.921;
   1:  PR[91,3] = PR[90,3] + 12.275;
   1:L PR[91] R[100]mm/sec CNT100;
   1:  PR[91,1] = PR[90,1] + 36.152;
   1:  PR[91,2] = PR[90,2] + -2.101;
   1:  PR[91,3] = PR[90,3] + 12.280;
   1:L PR[91] R[100]mm/sec CNT100;
   1:  PR[91,1] = PR[90,1] + 36.256;
   1:  PR[91,2] = PR[90,2] + -1.270;
   1:  PR[91,3] = PR[90,3] + 12.286;
   1:L PR[91] R[100]mm/sec CNT100;
   1:  PR[91,1] = PR[90,1] + 36.318;
   1:  PR[91,2] = PR[90,2] + -0.427;
   1:  PR[91,3] = PR[90,3] + 12.291;
   1:L PR[91] R[100]mm/sec CNT100;
   1:  PR[91,1] = PR[90,1] + 36.339;
   1:  PR[91,2] = PR[90,2] + 0.428;
   1:  PR[91,3] = PR[90,3] + 12.297;
   1:L PR[91] R[100]mm/sec CNT100;
   1:  PR[91,1] = PR[90,1] + 36.318;
   1:  PR[91,2] = PR[90,2] + 1.282;
   1:  PR[91,3] = PR[90,3] + 12.302;
   1:L PR[91] R[100]mm/sec CNT100;
   1:  PR[91,1] = PR[90,1] + 36.256;
   1:  PR[91,2] = PR[90,2] + 2.125;
   1:  PR[91,3] = PR[90,3] + 12.308;
   1:L PR[91] R[100]mm/sec CNT100;
   1:  PR[91,1] = PR[90,1] + 36.152;
   1:  PR[91,2] = PR[90,2] + 2.956;
   1:  PR[91,3] = PR[90,3] + 12.313;
   1:L PR[91] R[100]mm/sec CNT100;
   1:  PR[91,1] = PR[90,1] + 36.008;
   1:  PR[91,2] = PR[90,2] + 3.776;
   1:  PR[91,3] = PR[90,3] + 12.319;
   1:L PR[91] R[100]mm/sec CNT100;
   1:  PR[91,1] = PR[90,1] + 35.822;
   1:  PR[91,2] = PR[90,2] + 4.584;
   1:  PR[91,3] = PR[90,3] + 12.324;
   1:L PR[91] R[100]mm/sec CNT100;
   1:  PR[91,1] = PR[90,1] + 35.596;
   1:  PR[91,2] = PR[90,2] + 5.383;
   1:  PR[91,3] = PR[90,3] + 12.329;
   1:L PR[91] R[100]mm/sec CNT100;
   1:  PR[91,1] = PR[90,1] + 35.331;
   1:  PR[91,2] = PR[90,2] + 6.170;
   1:  PR[91,3] = PR[90,3] + 12.335;
   1:L PR[91] R[100]mm/sec CNT100;
   1:  PR[91,1] = PR[90,1] + 35.025;
   1:  PR[91,2] = PR[90,2] + 6.946;
   1:  PR[91,3] = PR[90,3] + 12.340;
   1:L PR[91] R[100]mm/sec CNT100;
   1:  PR[91,1] = PR[90,1] + 34.676;
   1:  PR[91,2] = PR[90,2] + 7.719;
   1:  PR[91,3] = PR[90,3] + 12.345;
   1:L PR[91] R[100]mm/sec CNT100;
   1:  PR[91,1] = PR[90,1] + 34.294;
   1:  PR[91,2] = PR[90,2] + 8.466;
   1:  PR[91,3] = PR[90,3] + 12.351;
   1:L PR[91] R[100]mm/sec CNT100;
   1:  PR[91,1] = PR[90,1] + 33.883;
   1:  PR[91,2] = PR[90,2] + 9.182;
   1:  PR[91,3] = PR[90,3] + 12.356;
   1:L PR[91] R[100]mm/sec CNT100;
   1:  PR[91,1] = PR[90,1] + 33.431;
   1:  PR[91,2] = PR[90,2] + 9.888;
   1:  PR[91,3] = PR[90,3] + 12.362;
   1:L PR[91] R[100]mm/sec CNT100;
   1:  PR[91,1] = PR[90,1] + 32.945;
   1:  PR[91,2] = PR[90,2] + 10.570;
   1:  PR[91,3] = PR[90,3] + 12.367;
   1:L PR[91] R[100]mm/sec CNT100;
   1:  PR[91,1] = PR[90,1] + 32.428;
   1:  PR[91,2] = PR[90,2] + 11.225;
   1:  PR[91,3] = PR[90,3] + 12.372;
   1:L PR[91] R[100]mm/sec CNT100;
   1:  PR[91,1] = PR[90,1] + 31.759;
   1:  PR[91,2] = PR[90,2] + 11.982;
   1:  PR[91,3] = PR[90,3] + 12.378;
   1:L PR[91] R[100]mm/sec CNT100;
   1:  PR[91,1] = PR[90,1] + 31.300;
   1:  PR[91,2] = PR[90,2] + 12.457;
   1:  PR[91,3] = PR[90,3] + 12.384;
   1:L PR[91] R[100]mm/sec CNT100;
   1:  PR[91,1] = PR[90,1] + 30.693;
   1:  PR[91,2] = PR[90,2] + 13.028;
   1:  PR[91,3] = PR[90,3] + 12.388;
   1:L PR[91] R[100]mm/sec CNT100;
   1:  PR[91,1] = PR[90,1] + 30.060;
   1:  PR[91,2] = PR[90,2] + 13.568;
   1:  PR[91,3] = PR[90,3] + 12.394;
   1:L PR[91] R[100]mm/sec CNT100;
   1:  PR[91,1] = PR[90,1] + 29.401;
   1:  PR[91,2] = PR[90,2] + 14.078;
   1:  PR[91,3] = PR[90,3] + 12.399;
   1:L PR[91] R[100]mm/sec CNT100;
   1:  PR[91,1] = PR[90,1] + 29.123;
   1:  PR[91,2] = PR[90,2] + 14.275;
   1:  PR[91,3] = PR[90,3] + 12.405;
   1:L PR[91] R[100]mm/sec CNT100;
   1:  PR[91,1] = PR[90,1] + 28.724;
   1:  PR[91,2] = PR[90,2] + 14.551;
   1:  PR[91,3] = PR[90,3] + 12.407;
   1:L PR[91] R[100]mm/sec CNT100;
   1:  PR[91,1] = PR[90,1] + 28.021;
   1:  PR[91,2] = PR[90,2] + 14.993;
   1:  PR[91,3] = PR[90,3] + 12.410;
   1:L PR[91] R[100]mm/sec CNT100;
   1:  PR[91,1] = PR[90,1] + 27.298;
   1:  PR[91,2] = PR[90,2] + 15.401;
   1:  PR[91,3] = PR[90,3] + 12.415;
   1:L PR[91] R[100]mm/sec CNT100;
   1:  PR[91,1] = PR[90,1] + 26.857;
   1:  PR[91,2] = PR[90,2] + 15.626;
   1:  PR[91,3] = PR[90,3] + 12.421;
   1:L PR[91] R[100]mm/sec CNT100;
   1:  PR[91,1] = PR[90,1] + 25.804;
   1:  PR[91,2] = PR[90,2] + 16.109;
   1:  PR[91,3] = PR[90,3] + 12.424;
   1:L PR[91] R[100]mm/sec CNT100;
   1:  PR[91,1] = PR[90,1] + 25.038;
   1:  PR[91,2] = PR[90,2] + 16.408;
   1:  PR[91,3] = PR[90,3] + 12.431;
   1:L PR[91] R[100]mm/sec CNT100;
   1:  PR[91,1] = PR[90,1] + 24.392;
   1:  PR[91,2] = PR[90,2] + 16.628;
   1:  PR[91,3] = PR[90,3] + 12.437;
   1:L PR[91] R[100]mm/sec CNT100;
   1:  PR[91,1] = PR[90,1] + 23.469;
   1:  PR[91,2] = PR[90,2] + 16.897;
   1:  PR[91,3] = PR[90,3] + 12.441;
   1:L PR[91] R[100]mm/sec CNT100;
   1:  PR[91,1] = PR[90,1] + 22.660;
   1:  PR[91,2] = PR[90,2] + 17.087;
   1:  PR[91,3] = PR[90,3] + 12.447;
   1:L PR[91] R[100]mm/sec CNT100;
   1:  PR[91,1] = PR[90,1] + 21.834;
   1:  PR[91,2] = PR[90,2] + 17.241;
   1:  PR[91,3] = PR[90,3] + 12.453;
   1:L PR[91] R[100]mm/sec CNT100;
   1:  PR[91,1] = PR[90,1] + 20.986;
   1:  PR[91,2] = PR[90,2] + 17.357;
   1:  PR[91,3] = PR[90,3] + 12.458;
   1:L PR[91] R[100]mm/sec CNT100;
   1:  PR[91,1] = PR[90,1] + 20.132;
   1:  PR[91,2] = PR[90,2] + 17.431;
   1:  PR[91,3] = PR[90,3] + 12.463;
   1:L PR[91] R[100]mm/sec CNT100;
   1:  PR[91,1] = PR[90,1] + 19.274;
   1:  PR[91,2] = PR[90,2] + 17.465;
   1:  PR[91,3] = PR[90,3] + 12.469;
   1:L PR[91] R[100]mm/sec CNT100;
   1:  PR[91,1] = PR[90,1] + 18.414;
   1:  PR[91,2] = PR[90,2] + 17.456;
   1:  PR[91,3] = PR[90,3] + 12.475;
   1:L PR[91] R[100]mm/sec CNT100;
   1:  PR[91,1] = PR[90,1] + 17.553;
   1:  PR[91,2] = PR[90,2] + 17.407;
   1:  PR[91,3] = PR[90,3] + 12.480;
   1:L PR[91] R[100]mm/sec CNT100;
   1:  PR[91,1] = PR[90,1] + 17.197;
   1:  PR[91,2] = PR[90,2] + 17.370;
   1:  PR[91,3] = PR[90,3] + 12.486;
   1:L PR[91] R[100]mm/sec CNT100;
   1:  PR[91,1] = PR[90,1] + 16.697;
   1:  PR[91,2] = PR[90,2] + 17.315;
   1:  PR[91,3] = PR[90,3] + 12.488;
   1:L PR[91] R[100]mm/sec CNT100;
   1:  PR[91,1] = PR[90,1] + 15.842;
   1:  PR[91,2] = PR[90,2] + 17.181;
   1:  PR[91,3] = PR[90,3] + 12.491;
   1:L PR[91] R[100]mm/sec CNT100;
   1:  PR[91,1] = PR[90,1] + 14.995;
   1:  PR[91,2] = PR[90,2] + 17.006;
   1:  PR[91,3] = PR[90,3] + 12.497;
   1:L PR[91] R[100]mm/sec CNT100;
   1:  PR[91,1] = PR[90,1] + 14.155;
   1:  PR[91,2] = PR[90,2] + 16.789;
   1:  PR[91,3] = PR[90,3] + 12.502;
   1:L PR[91] R[100]mm/sec CNT100;
   1:  PR[91,1] = PR[90,1] + 13.324;
   1:  PR[91,2] = PR[90,2] + 16.531;
   1:  PR[91,3] = PR[90,3] + 12.508;
   1:L PR[91] R[100]mm/sec CNT100;
   1:  PR[91,1] = PR[90,1] + 12.504;
   1:  PR[91,2] = PR[90,2] + 16.233;
   1:  PR[91,3] = PR[90,3] + 12.514;
   1:L PR[91] R[100]mm/sec CNT100;
   1:  PR[91,1] = PR[90,1] + 11.699;
   1:  PR[91,2] = PR[90,2] + 15.895;
   1:  PR[91,3] = PR[90,3] + 12.519;
   1:L PR[91] R[100]mm/sec CNT100;
   1:  PR[91,1] = PR[90,1] + 10.911;
   1:  PR[91,2] = PR[90,2] + 15.519;
   1:  PR[91,3] = PR[90,3] + 12.525;
   1:L PR[91] R[100]mm/sec CNT100;
   1:  PR[91,1] = PR[90,1] + 10.142;
   1:  PR[91,2] = PR[90,2] + 15.103;
   1:  PR[91,3] = PR[90,3] + 12.530;
   1:L PR[91] R[100]mm/sec CNT100;
   1:  PR[91,1] = PR[90,1] + 9.397;
   1:  PR[91,2] = PR[90,2] + 14.652;
   1:  PR[91,3] = PR[90,3] + 12.536;
   1:L PR[91] R[100]mm/sec CNT100;
   1:  PR[91,1] = PR[90,1] + 8.481;
   1:  PR[91,2] = PR[90,2] + 14.021;
   1:  PR[91,3] = PR[90,3] + 12.542;
   1:L PR[91] R[100]mm/sec CNT100;
   1:  PR[91,1] = PR[90,1] + 7.972;
   1:  PR[91,2] = PR[90,2] + 13.638;
   1:  PR[91,3] = PR[90,3] + 12.549;
   1:L PR[91] R[100]mm/sec CNT100;
   1:  PR[91,1] = PR[90,1] + 7.300;
   1:  PR[91,2] = PR[90,2] + 13.078;
   1:  PR[91,3] = PR[90,3] + 12.553;
   1:L PR[91] R[100]mm/sec CNT100;
   1:  PR[91,1] = PR[90,1] + 6.657;
   1:  PR[91,2] = PR[90,2] + 12.485;
   1:  PR[91,3] = PR[90,3] + 12.559;
   1:L PR[91] R[100]mm/sec CNT100;
   1:  PR[91,1] = PR[90,1] + 6.110;
   1:  PR[91,2] = PR[90,2] + 11.930;
   1:  PR[91,3] = PR[90,3] + 12.564;
   1:L PR[91] R[100]mm/sec CNT100;
   1:  PR[91,1] = PR[90,1] + 5.460;
   1:  PR[91,2] = PR[90,2] + 11.202;
   1:  PR[91,3] = PR[90,3] + 12.569;
   1:L PR[91] R[100]mm/sec CNT100;
   1:  PR[91,1] = PR[90,1] + 4.914;
   1:  PR[91,2] = PR[90,2] + 10.517;
   1:  PR[91,3] = PR[90,3] + 12.576;
   1:L PR[91] R[100]mm/sec CNT100;
   1:  PR[91,1] = PR[90,1] + 4.402;
   1:  PR[91,2] = PR[90,2] + 9.803;
   1:  PR[91,3] = PR[90,3] + 12.581;
   1:L PR[91] R[100]mm/sec CNT100;
   1:  PR[91,1] = PR[90,1] + 4.142;
   1:  PR[91,2] = PR[90,2] + 9.403;
   1:  PR[91,3] = PR[90,3] + 12.587;
   1:L PR[91] R[100]mm/sec CNT100;
   1:  PR[91,1] = PR[90,1] + 3.719;
   1:  PR[91,2] = PR[90,2] + 8.708;
   1:  PR[91,3] = PR[90,3] + 12.590;
   1:L PR[91] R[100]mm/sec CNT100;
   1:  PR[91,1] = PR[90,1] + 3.329;
   1:  PR[91,2] = PR[90,2] + 7.994;
   1:  PR[91,3] = PR[90,3] + 12.595;
   1:L PR[91] R[100]mm/sec CNT100;
   1:  PR[91,1] = PR[90,1] + 3.101;
   1:  PR[91,2] = PR[90,2] + 7.542;
   1:  PR[91,3] = PR[90,3] + 12.600;
   1:L PR[91] R[100]mm/sec CNT100;
   1:  PR[91,1] = PR[90,1] + 2.478;
   1:  PR[91,2] = PR[90,2] + 6.145;
   1:  PR[91,3] = PR[90,3] + 12.604;
   1:L PR[91] R[100]mm/sec CNT100;
   1:  PR[91,1] = PR[90,1] + 2.256;
   1:  PR[91,2] = PR[90,2] + 5.776;
   1:  PR[91,3] = PR[90,3] + 12.614;
   1:L PR[91] R[100]mm/sec CNT100;
   1:  PR[91,1] = PR[90,1] + 1.999;
   1:  PR[91,2] = PR[90,2] + 5.442;
   1:  PR[91,3] = PR[90,3] + 12.616;
   1:L PR[91] R[100]mm/sec CNT100;
   1:  PR[91,1] = PR[90,1] + 1.714;
   1:  PR[91,2] = PR[90,2] + 5.152;
   1:  PR[91,3] = PR[90,3] + 12.619;
   1:L PR[91] R[100]mm/sec CNT100;
   1:  PR[91,1] = PR[90,1] + 1.543;
   1:  PR[91,2] = PR[90,2] + 5.010;
   1:  PR[91,3] = PR[90,3] + 12.622;
   1:L PR[91] R[100]mm/sec CNT100;
   1:  PR[91,1] = PR[90,1] + 1.373;
   1:  PR[91,2] = PR[90,2] + 4.885;
   1:  PR[91,3] = PR[90,3] + 12.623;
   1:L PR[91] R[100]mm/sec CNT100;
   1:  PR[91,1] = PR[90,1] + 1.025;
   1:  PR[91,2] = PR[90,2] + 4.683;
   1:  PR[91,3] = PR[90,3] + 12.624;
   1:L PR[91] R[100]mm/sec CNT100;
   1:  PR[91,1] = PR[90,1] + 0.648;
   1:  PR[91,2] = PR[90,2] + 4.533;
   1:  PR[91,3] = PR[90,3] + 12.627;
   1:L PR[91] R[100]mm/sec CNT100;
   1:  PR[91,1] = PR[90,1] + 0.341;
   1:  PR[91,2] = PR[90,2] + 4.457;
   1:  PR[91,3] = PR[90,3] + 12.630;
   1:L PR[91] R[100]mm/sec CNT100;
   1:  PR[91,1] = PR[90,1] + -0.165;
   1:  PR[91,2] = PR[90,2] + 4.415;
   1:  PR[91,3] = PR[90,3] + 12.632;
   1:L PR[91] R[100]mm/sec CNT100;
   1:  PR[91,1] = PR[90,1] + -0.489;
   1:  PR[91,2] = PR[90,2] + 4.442;
   1:  PR[91,3] = PR[90,3] + 12.635;
   1:L PR[91] R[100]mm/sec CNT100;
   1:  PR[91,1] = PR[90,1] + -0.896;
   1:  PR[91,2] = PR[90,2] + 4.534;
   1:  PR[91,3] = PR[90,3] + 12.637;
   1:L PR[91] R[100]mm/sec CNT100;
   1:  PR[91,1] = PR[90,1] + -1.398;
   1:  PR[91,2] = PR[90,2] + 4.752;
   1:  PR[91,3] = PR[90,3] + 12.640;
   1:L PR[91] R[100]mm/sec CNT100;
   1:  PR[91,1] = PR[90,1] + -1.632;
   1:  PR[91,2] = PR[90,2] + 4.897;
   1:  PR[91,3] = PR[90,3] + 12.643;
   1:L PR[91] R[100]mm/sec CNT100;
   1:  PR[91,1] = PR[90,1] + -1.952;
   1:  PR[91,2] = PR[90,2] + 5.148;
   1:  PR[91,3] = PR[90,3] + 12.645;
   1:L PR[91] R[100]mm/sec CNT100;
   1:  PR[91,1] = PR[90,1] + -2.241;
   1:  PR[91,2] = PR[90,2] + 5.443;
   1:  PR[91,3] = PR[90,3] + 12.648;
   1:L PR[91] R[100]mm/sec CNT100;
   1:  PR[91,1] = PR[90,1] + -2.442;
   1:  PR[91,2] = PR[90,2] + 5.698;
   1:  PR[91,3] = PR[90,3] + 12.650;
   1:L PR[91] R[100]mm/sec CNT100;
   1:  PR[91,1] = PR[90,1] + -2.720;
   1:  PR[91,2] = PR[90,2] + 6.145;
   1:  PR[91,3] = PR[90,3] + 12.652;
   1:L PR[91] R[100]mm/sec CNT100;
   1:  PR[91,1] = PR[90,1] + -3.345;
   1:  PR[91,2] = PR[90,2] + 7.552;
   1:  PR[91,3] = PR[90,3] + 12.656;
   1:L PR[91] R[100]mm/sec CNT100;
   1:  PR[91,1] = PR[90,1] + -3.576;
   1:  PR[91,2] = PR[90,2] + 8.011;
   1:  PR[91,3] = PR[90,3] + 12.666;
   1:L PR[91] R[100]mm/sec CNT100;
   1:  PR[91,1] = PR[90,1] + -3.738;
   1:  PR[91,2] = PR[90,2] + 8.324;
   1:  PR[91,3] = PR[90,3] + 12.669;
   1:L PR[91] R[100]mm/sec CNT100;
   1:  PR[91,1] = PR[90,1] + -4.174;
   1:  PR[91,2] = PR[90,2] + 9.083;
   1:  PR[91,3] = PR[90,3] + 12.671;
   1:L PR[91] R[100]mm/sec CNT100;
   1:  PR[91,1] = PR[90,1] + -4.647;
   1:  PR[91,2] = PR[90,2] + 9.820;
   1:  PR[91,3] = PR[90,3] + 12.677;
   1:L PR[91] R[100]mm/sec CNT100;
   1:  PR[91,1] = PR[90,1] + -5.158;
   1:  PR[91,2] = PR[90,2] + 10.531;
   1:  PR[91,3] = PR[90,3] + 12.683;
   1:L PR[91] R[100]mm/sec CNT100;
   1:  PR[91,1] = PR[90,1] + -5.705;
   1:  PR[91,2] = PR[90,2] + 11.214;
   1:  PR[91,3] = PR[90,3] + 12.688;
   1:L PR[91] R[100]mm/sec CNT100;
   1:  PR[91,1] = PR[90,1] + -6.287;
   1:  PR[91,2] = PR[90,2] + 11.868;
   1:  PR[91,3] = PR[90,3] + 12.694;
   1:L PR[91] R[100]mm/sec CNT100;
   1:  PR[91,1] = PR[90,1] + -6.913;
   1:  PR[91,2] = PR[90,2] + 12.502;
   1:  PR[91,3] = PR[90,3] + 12.700;
   1:L PR[91] R[100]mm/sec CNT100;
   1:  PR[91,1] = PR[90,1] + -7.545;
   1:  PR[91,2] = PR[90,2] + 13.083;
   1:  PR[91,3] = PR[90,3] + 12.705;
   1:L PR[91] R[100]mm/sec CNT100;
   1:  PR[91,1] = PR[90,1] + -8.217;
   1:  PR[91,2] = PR[90,2] + 13.641;
   1:  PR[91,3] = PR[90,3] + 12.711;
   1:L PR[91] R[100]mm/sec CNT100;
   1:  PR[91,1] = PR[90,1] + -8.917;
   1:  PR[91,2] = PR[90,2] + 14.165;
   1:  PR[91,3] = PR[90,3] + 12.716;
   1:L PR[91] R[100]mm/sec CNT100;
   1:  PR[91,1] = PR[90,1] + -9.379;
   1:  PR[91,2] = PR[90,2] + 14.480;
   1:  PR[91,3] = PR[90,3] + 12.722;
   1:L PR[91] R[100]mm/sec CNT100;
   1:  PR[91,1] = PR[90,1] + -9.639;
   1:  PR[91,2] = PR[90,2] + 14.653;
   1:  PR[91,3] = PR[90,3] + 12.726;
   1:L PR[91] R[100]mm/sec CNT100;
   1:  PR[91,1] = PR[90,1] + -10.385;
   1:  PR[91,2] = PR[90,2] + 15.105;
   1:  PR[91,3] = PR[90,3] + 12.728;
   1:L PR[91] R[100]mm/sec CNT100;
   1:  PR[91,1] = PR[90,1] + -11.432;
   1:  PR[91,2] = PR[90,2] + 15.655;
   1:  PR[91,3] = PR[90,3] + 12.733;
   1:L PR[91] R[100]mm/sec CNT100;
   1:  PR[91,1] = PR[90,1] + -11.944;
   1:  PR[91,2] = PR[90,2] + 15.899;
   1:  PR[91,3] = PR[90,3] + 12.741;
   1:L PR[91] R[100]mm/sec CNT100;
   1:  PR[91,1] = PR[90,1] + -12.750;
   1:  PR[91,2] = PR[90,2] + 16.237;
   1:  PR[91,3] = PR[90,3] + 12.745;
   1:L PR[91] R[100]mm/sec CNT100;
   1:  PR[91,1] = PR[90,1] + -13.569;
   1:  PR[91,2] = PR[90,2] + 16.535;
   1:  PR[91,3] = PR[90,3] + 12.750;
   1:L PR[91] R[100]mm/sec CNT100;
   1:  PR[91,1] = PR[90,1] + -14.400;
   1:  PR[91,2] = PR[90,2] + 16.792;
   1:  PR[91,3] = PR[90,3] + 12.756;
   1:L PR[91] R[100]mm/sec CNT100;
   1:  PR[91,1] = PR[90,1] + -15.239;
   1:  PR[91,2] = PR[90,2] + 17.008;
   1:  PR[91,3] = PR[90,3] + 12.761;
   1:L PR[91] R[100]mm/sec CNT100;
   1:  PR[91,1] = PR[90,1] + -16.086;
   1:  PR[91,2] = PR[90,2] + 17.182;
   1:  PR[91,3] = PR[90,3] + 12.767;
   1:L PR[91] R[100]mm/sec CNT100;
   1:  PR[91,1] = PR[90,1] + -16.940;
   1:  PR[91,2] = PR[90,2] + 17.315;
   1:  PR[91,3] = PR[90,3] + 12.773;
   1:L PR[91] R[100]mm/sec CNT100;
   1:  PR[91,1] = PR[90,1] + -17.798;
   1:  PR[91,2] = PR[90,2] + 17.407;
   1:  PR[91,3] = PR[90,3] + 12.778;
   1:L PR[91] R[100]mm/sec CNT100;
   1:  PR[91,1] = PR[90,1] + -18.659;
   1:  PR[91,2] = PR[90,2] + 17.457;
   1:  PR[91,3] = PR[90,3] + 12.784;
   1:L PR[91] R[100]mm/sec CNT100;
   1:  PR[91,1] = PR[90,1] + -19.004;
   1:  PR[91,2] = PR[90,2] + 17.461;
   1:  PR[91,3] = PR[90,3] + 12.789;
   1:L PR[91] R[100]mm/sec CNT100;
   1:  PR[91,1] = PR[90,1] + -19.517;
   1:  PR[91,2] = PR[90,2] + 17.465;
   1:  PR[91,3] = PR[90,3] + 12.792;
   1:L PR[91] R[100]mm/sec CNT100;
   1:  PR[91,1] = PR[90,1] + -20.375;
   1:  PR[91,2] = PR[90,2] + 17.431;
   1:  PR[91,3] = PR[90,3] + 12.795;
   1:L PR[91] R[100]mm/sec CNT100;
   1:  PR[91,1] = PR[90,1] + -21.229;
   1:  PR[91,2] = PR[90,2] + 17.356;
   1:  PR[91,3] = PR[90,3] + 12.800;
   1:L PR[91] R[100]mm/sec CNT100;
   1:  PR[91,1] = PR[90,1] + -22.076;
   1:  PR[91,2] = PR[90,2] + 17.240;
   1:  PR[91,3] = PR[90,3] + 12.806;
   1:L PR[91] R[100]mm/sec CNT100;
   1:  PR[91,1] = PR[90,1] + -22.916;
   1:  PR[91,2] = PR[90,2] + 17.084;
   1:  PR[91,3] = PR[90,3] + 12.811;
   1:L PR[91] R[100]mm/sec CNT100;
   1:  PR[91,1] = PR[90,1] + -23.780;
   1:  PR[91,2] = PR[90,2] + 16.878;
   1:  PR[91,3] = PR[90,3] + 12.817;
   1:L PR[91] R[100]mm/sec CNT100;
   1:  PR[91,1] = PR[90,1] + -24.634;
   1:  PR[91,2] = PR[90,2] + 16.628;
   1:  PR[91,3] = PR[90,3] + 12.823;
   1:L PR[91] R[100]mm/sec CNT100;
   1:  PR[91,1] = PR[90,1] + -25.280;
   1:  PR[91,2] = PR[90,2] + 16.408;
   1:  PR[91,3] = PR[90,3] + 12.828;
   1:L PR[91] R[100]mm/sec CNT100;
   1:  PR[91,1] = PR[90,1] + -26.048;
   1:  PR[91,2] = PR[90,2] + 16.108;
   1:  PR[91,3] = PR[90,3] + 12.833;
   1:L PR[91] R[100]mm/sec CNT100;
   1:  PR[91,1] = PR[90,1] + -26.802;
   1:  PR[91,2] = PR[90,2] + 15.771;
   1:  PR[91,3] = PR[90,3] + 12.838;
   1:L PR[91] R[100]mm/sec CNT100;
   1:  PR[91,1] = PR[90,1] + -27.542;
   1:  PR[91,2] = PR[90,2] + 15.398;
   1:  PR[91,3] = PR[90,3] + 12.843;
   1:L PR[91] R[100]mm/sec CNT100;
   1:  PR[91,1] = PR[90,1] + -27.872;
   1:  PR[91,2] = PR[90,2] + 15.214;
   1:  PR[91,3] = PR[90,3] + 12.849;
   1:L PR[91] R[100]mm/sec CNT100;
   1:  PR[91,1] = PR[90,1] + -28.260;
   1:  PR[91,2] = PR[90,2] + 14.992;
   1:  PR[91,3] = PR[90,3] + 12.851;
   1:L PR[91] R[100]mm/sec CNT100;
   1:  PR[91,1] = PR[90,1] + -28.963;
   1:  PR[91,2] = PR[90,2] + 14.549;
   1:  PR[91,3] = PR[90,3] + 12.854;
   1:L PR[91] R[100]mm/sec CNT100;
   1:  PR[91,1] = PR[90,1] + -29.643;
   1:  PR[91,2] = PR[90,2] + 14.074;
   1:  PR[91,3] = PR[90,3] + 12.859;
   1:L PR[91] R[100]mm/sec CNT100;
   1:  PR[91,1] = PR[90,1] + -30.300;
   1:  PR[91,2] = PR[90,2] + 13.566;
   1:  PR[91,3] = PR[90,3] + 12.865;
   1:L PR[91] R[100]mm/sec CNT100;
   1:  PR[91,1] = PR[90,1] + -30.934;
   1:  PR[91,2] = PR[90,2] + 13.026;
   1:  PR[91,3] = PR[90,3] + 12.870;
   1:L PR[91] R[100]mm/sec CNT100;
   1:  PR[91,1] = PR[90,1] + -31.385;
   1:  PR[91,2] = PR[90,2] + 12.603;
   1:  PR[91,3] = PR[90,3] + 12.876;
   1:L PR[91] R[100]mm/sec CNT100;
   1:  PR[91,1] = PR[90,1] + -32.119;
   1:  PR[91,2] = PR[90,2] + 11.854;
   1:  PR[91,3] = PR[90,3] + 12.880;
   1:L PR[91] R[100]mm/sec CNT100;
   1:  PR[91,1] = PR[90,1] + -32.667;
   1:  PR[91,2] = PR[90,2] + 11.227;
   1:  PR[91,3] = PR[90,3] + 12.886;
   1:L PR[91] R[100]mm/sec CNT100;
   1:  PR[91,1] = PR[90,1] + -33.184;
   1:  PR[91,2] = PR[90,2] + 10.572;
   1:  PR[91,3] = PR[90,3] + 12.892;
   1:L PR[91] R[100]mm/sec CNT100;
   1:  PR[91,1] = PR[90,1] + -33.670;
   1:  PR[91,2] = PR[90,2] + 9.890;
   1:  PR[91,3] = PR[90,3] + 12.897;
   1:L PR[91] R[100]mm/sec CNT100;
   1:  PR[91,1] = PR[90,1] + -34.121;
   1:  PR[91,2] = PR[90,2] + 9.184;
   1:  PR[91,3] = PR[90,3] + 12.902;
   1:L PR[91] R[100]mm/sec CNT100;
   1:  PR[91,1] = PR[90,1] + -34.538;
   1:  PR[91,2] = PR[90,2] + 8.457;
   1:  PR[91,3] = PR[90,3] + 12.908;
   1:L PR[91] R[100]mm/sec CNT100;
   1:  PR[91,1] = PR[90,1] + -34.920;
   1:  PR[91,2] = PR[90,2] + 7.709;
   1:  PR[91,3] = PR[90,3] + 12.913;
   1:L PR[91] R[100]mm/sec CNT100;
   1:  PR[91,1] = PR[90,1] + -35.264;
   1:  PR[91,2] = PR[90,2] + 6.944;
   1:  PR[91,3] = PR[90,3] + 12.919;
   1:L PR[91] R[100]mm/sec CNT100;
   1:  PR[91,1] = PR[90,1] + -35.569;
   1:  PR[91,2] = PR[90,2] + 6.166;
   1:  PR[91,3] = PR[90,3] + 12.924;
   1:L PR[91] R[100]mm/sec CNT100;
   1:  PR[91,1] = PR[90,1] + -35.835;
   1:  PR[91,2] = PR[90,2] + 5.377;
   1:  PR[91,3] = PR[90,3] + 12.929;
   1:L PR[91] R[100]mm/sec CNT100;
   1:  PR[91,1] = PR[90,1] + -36.061;
   1:  PR[91,2] = PR[90,2] + 4.578;
   1:  PR[91,3] = PR[90,3] + 12.935;
   1:L PR[91] R[100]mm/sec CNT100;
   1:  PR[91,1] = PR[90,1] + -36.246;
   1:  PR[91,2] = PR[90,2] + 3.770;
   1:  PR[91,3] = PR[90,3] + 12.940;
   1:L PR[91] R[100]mm/sec CNT100;
   1:  PR[91,1] = PR[90,1] + -36.391;
   1:  PR[91,2] = PR[90,2] + 2.952;
   1:  PR[91,3] = PR[90,3] + 12.945;
   1:L PR[91] R[100]mm/sec CNT100;
   1:  PR[91,1] = PR[90,1] + -36.495;
   1:  PR[91,2] = PR[90,2] + 2.123;
   1:  PR[91,3] = PR[90,3] + 12.951;
   1:L PR[91] R[100]mm/sec CNT100;
   1:  PR[91,1] = PR[90,1] + -36.557;
   1:  PR[91,2] = PR[90,2] + 1.281;
   1:  PR[91,3] = PR[90,3] + 12.956;
   1:L PR[91] R[100]mm/sec CNT100;
   1:  PR[91,1] = PR[90,1] + -36.578;
   1:  PR[91,2] = PR[90,2] + 0.428;
   1:  PR[91,3] = PR[90,3] + 12.962;
   1:L PR[91] R[100]mm/sec CNT100;
   1:  PR[91,1] = PR[90,1] + -36.557;
   1:  PR[91,2] = PR[90,2] + -0.426;
   1:  PR[91,3] = PR[90,3] + 12.967;
   1:L PR[91] R[100]mm/sec CNT100;
   1:  PR[91,1] = PR[90,1] + -36.495;
   1:  PR[91,2] = PR[90,2] + -1.268;
   1:  PR[91,3] = PR[90,3] + 12.973;
   1:L PR[91] R[100]mm/sec CNT100;
   1:  PR[91,1] = PR[90,1] + -36.391;
   1:  PR[91,2] = PR[90,2] + -2.097;
   1:  PR[91,3] = PR[90,3] + 12.978;
   1:L PR[91] R[100]mm/sec CNT100;
   1:  PR[91,1] = PR[90,1] + -36.246;
   1:  PR[91,2] = PR[90,2] + -2.915;
   1:  PR[91,3] = PR[90,3] + 12.984;
   1:L PR[91] R[100]mm/sec CNT100;
   1:  PR[91,1] = PR[90,1] + -36.061;
   1:  PR[91,2] = PR[90,2] + -3.723;
   1:  PR[91,3] = PR[90,3] + 12.989;
   1:L PR[91] R[100]mm/sec CNT100;
   1:  PR[91,1] = PR[90,1] + -35.835;
   1:  PR[91,2] = PR[90,2] + -4.522;
   1:  PR[91,3] = PR[90,3] + 12.994;
   1:L PR[91] R[100]mm/sec CNT100;
   1:  PR[91,1] = PR[90,1] + -35.569;
   1:  PR[91,2] = PR[90,2] + -5.311;
   1:  PR[91,3] = PR[90,3] + 13.000;
   1:L PR[91] R[100]mm/sec CNT100;
   1:  PR[91,1] = PR[90,1] + -35.264;
   1:  PR[91,2] = PR[90,2] + -6.089;
   1:  PR[91,3] = PR[90,3] + 13.005;
   1:L PR[91] R[100]mm/sec CNT100;
   1:  PR[91,1] = PR[90,1] + -34.915;
   1:  PR[91,2] = PR[90,2] + -6.864;
   1:  PR[91,3] = PR[90,3] + 13.010;
   1:L PR[91] R[100]mm/sec CNT100;
   1:  PR[91,1] = PR[90,1] + -34.532;
   1:  PR[91,2] = PR[90,2] + -7.613;
   1:  PR[91,3] = PR[90,3] + 13.016;
   1:L PR[91] R[100]mm/sec CNT100;
   1:  PR[91,1] = PR[90,1] + -34.121;
   1:  PR[91,2] = PR[90,2] + -8.329;
   1:  PR[91,3] = PR[90,3] + 13.021;
   1:L PR[91] R[100]mm/sec CNT100;
   1:  PR[91,1] = PR[90,1] + -33.670;
   1:  PR[91,2] = PR[90,2] + -9.035;
   1:  PR[91,3] = PR[90,3] + 13.027;
   1:L PR[91] R[100]mm/sec CNT100;
   1:  PR[91,1] = PR[90,1] + -33.184;
   1:  PR[91,2] = PR[90,2] + -9.716;
   1:  PR[91,3] = PR[90,3] + 13.032;
   1:L PR[91] R[100]mm/sec CNT100;
   1:  PR[91,1] = PR[90,1] + -32.667;
   1:  PR[91,2] = PR[90,2] + -10.372;
   1:  PR[91,3] = PR[90,3] + 13.037;
   1:L PR[91] R[100]mm/sec CNT100;
   1:  PR[91,1] = PR[90,1] + -32.119;
   1:  PR[91,2] = PR[90,2] + -10.999;
   1:  PR[91,3] = PR[90,3] + 13.043;
   1:L PR[91] R[100]mm/sec CNT100;
   1:  PR[91,1] = PR[90,1] + -31.385;
   1:  PR[91,2] = PR[90,2] + -11.748;
   1:  PR[91,3] = PR[90,3] + 13.048;
   1:L PR[91] R[100]mm/sec CNT100;
   1:  PR[91,1] = PR[90,1] + -30.934;
   1:  PR[91,2] = PR[90,2] + -12.171;
   1:  PR[91,3] = PR[90,3] + 13.055;
   1:L PR[91] R[100]mm/sec CNT100;
   1:  PR[91,1] = PR[90,1] + -30.300;
   1:  PR[91,2] = PR[90,2] + -12.711;
   1:  PR[91,3] = PR[90,3] + 13.059;
   1:L PR[91] R[100]mm/sec CNT100;
   1:  PR[91,1] = PR[90,1] + -29.641;
   1:  PR[91,2] = PR[90,2] + -13.220;
   1:  PR[91,3] = PR[90,3] + 13.064;
   1:L PR[91] R[100]mm/sec CNT100;
   1:  PR[91,1] = PR[90,1] + -29.364;
   1:  PR[91,2] = PR[90,2] + -13.417;
   1:  PR[91,3] = PR[90,3] + 13.070;
   1:L PR[91] R[100]mm/sec CNT100;
   1:  PR[91,1] = PR[90,1] + -28.964;
   1:  PR[91,2] = PR[90,2] + -13.693;
   1:  PR[91,3] = PR[90,3] + 13.072;
   1:L PR[91] R[100]mm/sec CNT100;
   1:  PR[91,1] = PR[90,1] + -28.261;
   1:  PR[91,2] = PR[90,2] + -14.136;
   1:  PR[91,3] = PR[90,3] + 13.075;
   1:L PR[91] R[100]mm/sec CNT100;
   1:  PR[91,1] = PR[90,1] + -27.539;
   1:  PR[91,2] = PR[90,2] + -14.544;
   1:  PR[91,3] = PR[90,3] + 13.080;
   1:L PR[91] R[100]mm/sec CNT100;
   1:  PR[91,1] = PR[90,1] + -27.098;
   1:  PR[91,2] = PR[90,2] + -14.770;
   1:  PR[91,3] = PR[90,3] + 13.086;
   1:L PR[91] R[100]mm/sec CNT100;
   1:  PR[91,1] = PR[90,1] + -26.045;
   1:  PR[91,2] = PR[90,2] + -15.254;
   1:  PR[91,3] = PR[90,3] + 13.089;
   1:L PR[91] R[100]mm/sec CNT100;
   1:  PR[91,1] = PR[90,1] + -25.280;
   1:  PR[91,2] = PR[90,2] + -15.553;
   1:  PR[91,3] = PR[90,3] + 13.096;
   1:L PR[91] R[100]mm/sec CNT100;
   1:  PR[91,1] = PR[90,1] + -24.635;
   1:  PR[91,2] = PR[90,2] + -15.772;
   1:  PR[91,3] = PR[90,3] + 13.102;
   1:L PR[91] R[100]mm/sec CNT100;
   1:  PR[91,1] = PR[90,1] + -23.711;
   1:  PR[91,2] = PR[90,2] + -16.041;
   1:  PR[91,3] = PR[90,3] + 13.106;
   1:L PR[91] R[100]mm/sec CNT100;
   1:  PR[91,1] = PR[90,1] + -22.899;
   1:  PR[91,2] = PR[90,2] + -16.232;
   1:  PR[91,3] = PR[90,3] + 13.112;
   1:L PR[91] R[100]mm/sec CNT100;
   1:  PR[91,1] = PR[90,1] + -22.076;
   1:  PR[91,2] = PR[90,2] + -16.385;
   1:  PR[91,3] = PR[90,3] + 13.118;
   1:L PR[91] R[100]mm/sec CNT100;
   1:  PR[91,1] = PR[90,1] + -21.229;
   1:  PR[91,2] = PR[90,2] + -16.501;
   1:  PR[91,3] = PR[90,3] + 13.123;
   1:L PR[91] R[100]mm/sec CNT100;
   1:  PR[91,1] = PR[90,1] + -20.375;
   1:  PR[91,2] = PR[90,2] + -16.576;
   1:  PR[91,3] = PR[90,3] + 13.128;
   1:L PR[91] R[100]mm/sec CNT100;
   1:  PR[91,1] = PR[90,1] + -19.798;
   1:  PR[91,2] = PR[90,2] + -16.600;
   1:  PR[91,3] = PR[90,3] + 13.134;
   1:L PR[91] R[100]mm/sec CNT100;
   1:  PR[91,1] = PR[90,1] + -18.654;
   1:  PR[91,2] = PR[90,2] + -16.601;
   1:  PR[91,3] = PR[90,3] + 13.138;
   1:L PR[91] R[100]mm/sec CNT100;
   1:  PR[91,1] = PR[90,1] + -17.801;
   1:  PR[91,2] = PR[90,2] + -16.552;
   1:  PR[91,3] = PR[90,3] + 13.145;
   1:L PR[91] R[100]mm/sec CNT100;
   1:  PR[91,1] = PR[90,1] + -16.655;
   1:  PR[91,2] = PR[90,2] + -16.417;
   1:  PR[91,3] = PR[90,3] + 13.151;
   1:L PR[91] R[100]mm/sec CNT100;
   1:  PR[91,1] = PR[90,1] + -16.087;
   1:  PR[91,2] = PR[90,2] + -16.327;
   1:  PR[91,3] = PR[90,3] + 13.158;
   1:L PR[91] R[100]mm/sec CNT100;
   1:  PR[91,1] = PR[90,1] + -15.239;
   1:  PR[91,2] = PR[90,2] + -16.153;
   1:  PR[91,3] = PR[90,3] + 13.162;
   1:L PR[91] R[100]mm/sec CNT100;
   1:  PR[91,1] = PR[90,1] + -14.400;
   1:  PR[91,2] = PR[90,2] + -15.937;
   1:  PR[91,3] = PR[90,3] + 13.167;
   1:L PR[91] R[100]mm/sec CNT100;
   1:  PR[91,1] = PR[90,1] + -13.569;
   1:  PR[91,2] = PR[90,2] + -15.680;
   1:  PR[91,3] = PR[90,3] + 13.173;
   1:L PR[91] R[100]mm/sec CNT100;
   1:  PR[91,1] = PR[90,1] + -12.750;
   1:  PR[91,2] = PR[90,2] + -15.382;
   1:  PR[91,3] = PR[90,3] + 13.178;
   1:L PR[91] R[100]mm/sec CNT100;
   1:  PR[91,1] = PR[90,1] + -11.945;
   1:  PR[91,2] = PR[90,2] + -15.044;
   1:  PR[91,3] = PR[90,3] + 13.184;
   1:L PR[91] R[100]mm/sec CNT100;
   1:  PR[91,1] = PR[90,1] + -11.157;
   1:  PR[91,2] = PR[90,2] + -14.667;
   1:  PR[91,3] = PR[90,3] + 13.190;
   1:L PR[91] R[100]mm/sec CNT100;
   1:  PR[91,1] = PR[90,1] + -10.387;
   1:  PR[91,2] = PR[90,2] + -14.251;
   1:  PR[91,3] = PR[90,3] + 13.195;
   1:L PR[91] R[100]mm/sec CNT100;
   1:  PR[91,1] = PR[90,1] + -10.043;
   1:  PR[91,2] = PR[90,2] + -14.045;
   1:  PR[91,3] = PR[90,3] + 13.201;
   1:L PR[91] R[100]mm/sec CNT100;
   1:  PR[91,1] = PR[90,1] + -9.641;
   1:  PR[91,2] = PR[90,2] + -13.799;
   1:  PR[91,3] = PR[90,3] + 13.204;
   1:L PR[91] R[100]mm/sec CNT100;
   1:  PR[91,1] = PR[90,1] + -8.916;
   1:  PR[91,2] = PR[90,2] + -13.310;
   1:  PR[91,3] = PR[90,3] + 13.207;
   1:L PR[91] R[100]mm/sec CNT100;
   1:  PR[91,1] = PR[90,1] + -8.217;
   1:  PR[91,2] = PR[90,2] + -12.786;
   1:  PR[91,3] = PR[90,3] + 13.212;
   1:L PR[91] R[100]mm/sec CNT100;
   1:  PR[91,1] = PR[90,1] + -7.545;
   1:  PR[91,2] = PR[90,2] + -12.228;
   1:  PR[91,3] = PR[90,3] + 13.218;
   1:L PR[91] R[100]mm/sec CNT100;
   1:  PR[91,1] = PR[90,1] + -6.902;
   1:  PR[91,2] = PR[90,2] + -11.637;
   1:  PR[91,3] = PR[90,3] + 13.224;
   1:L PR[91] R[100]mm/sec CNT100;
   1:  PR[91,1] = PR[90,1] + -6.287;
   1:  PR[91,2] = PR[90,2] + -11.013;
   1:  PR[91,3] = PR[90,3] + 13.229;
   1:L PR[91] R[100]mm/sec CNT100;
   1:  PR[91,1] = PR[90,1] + -5.705;
   1:  PR[91,2] = PR[90,2] + -10.359;
   1:  PR[91,3] = PR[90,3] + 13.235;
   1:L PR[91] R[100]mm/sec CNT100;
   1:  PR[91,1] = PR[90,1] + -5.158;
   1:  PR[91,2] = PR[90,2] + -9.676;
   1:  PR[91,3] = PR[90,3] + 13.240;
   1:L PR[91] R[100]mm/sec CNT100;
   1:  PR[91,1] = PR[90,1] + -4.647;
   1:  PR[91,2] = PR[90,2] + -8.965;
   1:  PR[91,3] = PR[90,3] + 13.246;
   1:L PR[91] R[100]mm/sec CNT100;
   1:  PR[91,1] = PR[90,1] + -4.173;
   1:  PR[91,2] = PR[90,2] + -8.227;
   1:  PR[91,3] = PR[90,3] + 13.252;
   1:L PR[91] R[100]mm/sec CNT100;
   1:  PR[91,1] = PR[90,1] + -3.963;
   1:  PR[91,2] = PR[90,2] + -7.867;
   1:  PR[91,3] = PR[90,3] + 13.257;
   1:L PR[91] R[100]mm/sec CNT100;
   1:  PR[91,1] = PR[90,1] + -3.740;
   1:  PR[91,2] = PR[90,2] + -7.472;
   1:  PR[91,3] = PR[90,3] + 13.260;
   1:L PR[91] R[100]mm/sec CNT100;
   1:  PR[91,1] = PR[90,1] + -3.344;
   1:  PR[91,2] = PR[90,2] + -6.696;
   1:  PR[91,3] = PR[90,3] + 13.263;
   1:L PR[91] R[100]mm/sec CNT100;
   1:  PR[91,1] = PR[90,1] + -2.721;
   1:  PR[91,2] = PR[90,2] + -5.293;
   1:  PR[91,3] = PR[90,3] + 13.269;
   1:L PR[91] R[100]mm/sec CNT100;
   1:  PR[91,1] = PR[90,1] + -2.499;
   1:  PR[91,2] = PR[90,2] + -4.923;
   1:  PR[91,3] = PR[90,3] + 13.279;
   1:L PR[91] R[100]mm/sec CNT100;
   1:  PR[91,1] = PR[90,1] + -2.242;
   1:  PR[91,2] = PR[90,2] + -4.589;
   1:  PR[91,3] = PR[90,3] + 13.281;
   1:L PR[91] R[100]mm/sec CNT100;
   1:  PR[91,1] = PR[90,1] + -1.950;
   1:  PR[91,2] = PR[90,2] + -4.291;
   1:  PR[91,3] = PR[90,3] + 13.284;
   1:L PR[91] R[100]mm/sec CNT100;
   1:  PR[91,1] = PR[90,1] + -1.624;
   1:  PR[91,2] = PR[90,2] + -4.036;
   1:  PR[91,3] = PR[90,3] + 13.287;
   1:L PR[91] R[100]mm/sec CNT100;
   1:  PR[91,1] = PR[90,1] + -1.274;
   1:  PR[91,2] = PR[90,2] + -3.832;
   1:  PR[91,3] = PR[90,3] + 13.289;
   1:L PR[91] R[100]mm/sec CNT100;
   1:  PR[91,1] = PR[90,1] + -1.000;
   1:  PR[91,2] = PR[90,2] + -3.715;
   1:  PR[91,3] = PR[90,3] + 13.292;
   1:L PR[91] R[100]mm/sec CNT100;
   1:  PR[91,1] = PR[90,1] + -0.488;
   1:  PR[91,2] = PR[90,2] + -3.585;
   1:  PR[91,3] = PR[90,3] + 13.294;
   1:L PR[91] R[100]mm/sec CNT100;
   1:  PR[91,1] = PR[90,1] + -0.070;
   1:  PR[91,2] = PR[90,2] + -3.560;
   1:  PR[91,3] = PR[90,3] + 13.297;
   1:L PR[91] R[100]mm/sec CNT100;
   1:  PR[91] = PR[90];
   1:  PR[91,1] = PR[90,1] + 0.202;
   1:  PR[91,2] = PR[90,2] + -4.645;
   1:  PR[91,3] = PR[90,3] + 14.630;
   1:L PR[91] R[100]mm/sec CNT100;
   1:  PR[91,1] = PR[90,1] + 0.610;
   1:  PR[91,2] = PR[90,2] + -4.731;
   1:  PR[91,3] = PR[90,3] + 13.303;
   1:L PR[91] R[100]mm/sec CNT100;
   1:  PR[91,1] = PR[90,1] + 0.809;
   1:  PR[91,2] = PR[90,2] + -4.798;
   1:  PR[91,3] = PR[90,3] + 13.305;
   1:L PR[91] R[100]mm/sec CNT100;
   1:  PR[91,1] = PR[90,1] + 1.176;
   1:  PR[91,2] = PR[90,2] + -4.968;
   1:  PR[91,3] = PR[90,3] + 13.307;
   1:L PR[91] R[100]mm/sec CNT100;
   1:  PR[91,1] = PR[90,1] + 1.522;
   1:  PR[91,2] = PR[90,2] + -5.195;
   1:  PR[91,3] = PR[90,3] + 13.309;
   1:L PR[91] R[100]mm/sec CNT100;
   1:  PR[91,1] = PR[90,1] + 1.787;
   1:  PR[91,2] = PR[90,2] + -5.420;
   1:  PR[91,3] = PR[90,3] + 13.312;
   1:L PR[91] R[100]mm/sec CNT100;
   1:  PR[91,1] = PR[90,1] + 2.105;
   1:  PR[91,2] = PR[90,2] + -5.766;
   1:  PR[91,3] = PR[90,3] + 13.314;
   1:L PR[91] R[100]mm/sec CNT100;
   1:  PR[91,1] = PR[90,1] + 2.387;
   1:  PR[91,2] = PR[90,2] + -6.171;
   1:  PR[91,3] = PR[90,3] + 13.318;
   1:L PR[91] R[100]mm/sec CNT100;
   1:  PR[91,1] = PR[90,1] + 2.885;
   1:  PR[91,2] = PR[90,2] + -7.152;
   1:  PR[91,3] = PR[90,3] + 13.321;
   1:L PR[91] R[100]mm/sec CNT100;
   1:  PR[91,1] = PR[90,1] + 3.320;
   1:  PR[91,2] = PR[90,2] + -7.936;
   1:  PR[91,3] = PR[90,3] + 13.328;
   1:L PR[91] R[100]mm/sec CNT100;
   1:  PR[91,1] = PR[90,1] + 3.772;
   1:  PR[91,2] = PR[90,2] + -8.667;
   1:  PR[91,3] = PR[90,3] + 13.334;
   1:L PR[91] R[100]mm/sec CNT100;
   1:  PR[91,1] = PR[90,1] + 4.192;
   1:  PR[91,2] = PR[90,2] + -9.280;
   1:  PR[91,3] = PR[90,3] + 13.339;
   1:L PR[91] R[100]mm/sec CNT100;
   1:  PR[91,1] = PR[90,1] + 4.817;
   1:  PR[91,2] = PR[90,2] + -10.104;
   1:  PR[91,3] = PR[90,3] + 13.344;
   1:L PR[91] R[100]mm/sec CNT100;
   1:  PR[91,1] = PR[90,1] + 5.184;
   1:  PR[91,2] = PR[90,2] + -10.538;
   1:  PR[91,3] = PR[90,3] + 13.351;
   1:L PR[91] R[100]mm/sec CNT100;
   1:  PR[91,1] = PR[90,1] + 6.014;
   1:  PR[91,2] = PR[90,2] + -11.432;
   1:  PR[91,3] = PR[90,3] + 13.355;
   1:L PR[91] R[100]mm/sec CNT100;
   1:  PR[91,1] = PR[90,1] + 6.894;
   1:  PR[91,2] = PR[90,2] + -12.251;
   1:  PR[91,3] = PR[90,3] + 13.363;
   1:L PR[91] R[100]mm/sec CNT100;
   1:  PR[91,1] = PR[90,1] + 7.356;
   1:  PR[91,2] = PR[90,2] + -12.639;
   1:  PR[91,3] = PR[90,3] + 13.371;
   1:L PR[91] R[100]mm/sec CNT100;
   1:  PR[91,1] = PR[90,1] + 8.080;
   1:  PR[91,2] = PR[90,2] + -13.195;
   1:  PR[91,3] = PR[90,3] + 13.375;
   1:L PR[91] R[100]mm/sec CNT100;
   1:  PR[91,1] = PR[90,1] + 8.833;
   1:  PR[91,2] = PR[90,2] + -13.713;
   1:  PR[91,3] = PR[90,3] + 13.381;
   1:L PR[91] R[100]mm/sec CNT100;
   1:  PR[91,1] = PR[90,1] + 9.591;
   1:  PR[91,2] = PR[90,2] + -14.182;
   1:  PR[91,3] = PR[90,3] + 13.387;
   1:L PR[91] R[100]mm/sec CNT100;
   1:  PR[91,1] = PR[90,1] + 10.179;
   1:  PR[91,2] = PR[90,2] + -14.509;
   1:  PR[91,3] = PR[90,3] + 13.392;
   1:L PR[91] R[100]mm/sec CNT100;
   1:  PR[91,1] = PR[90,1] + 11.172;
   1:  PR[91,2] = PR[90,2] + -15.004;
   1:  PR[91,3] = PR[90,3] + 13.397;
   1:L PR[91] R[100]mm/sec CNT100;
   1:  PR[91,1] = PR[90,1] + 11.988;
   1:  PR[91,2] = PR[90,2] + -15.354;
   1:  PR[91,3] = PR[90,3] + 13.404;
   1:L PR[91] R[100]mm/sec CNT100;
   1:  PR[91,1] = PR[90,1] + 12.819;
   1:  PR[91,2] = PR[90,2] + -15.664;
   1:  PR[91,3] = PR[90,3] + 13.410;
   1:L PR[91] R[100]mm/sec CNT100;
   1:  PR[91,1] = PR[90,1] + 13.839;
   1:  PR[91,2] = PR[90,2] + -15.980;
   1:  PR[91,3] = PR[90,3] + 13.416;
   1:L PR[91] R[100]mm/sec CNT100;
   1:  PR[91,1] = PR[90,1] + 14.524;
   1:  PR[91,2] = PR[90,2] + -16.161;
   1:  PR[91,3] = PR[90,3] + 13.423;
   1:L PR[91] R[100]mm/sec CNT100;
   1:  PR[91,1] = PR[90,1] + 15.390;
   1:  PR[91,2] = PR[90,2] + -16.346;
   1:  PR[91,3] = PR[90,3] + 13.427;
   1:L PR[91] R[100]mm/sec CNT100;
   1:  PR[91,1] = PR[90,1] + 16.258;
   1:  PR[91,2] = PR[90,2] + -16.488;
   1:  PR[91,3] = PR[90,3] + 13.433;
   1:L PR[91] R[100]mm/sec CNT100;
   1:  PR[91,1] = PR[90,1] + 17.131;
   1:  PR[91,2] = PR[90,2] + -16.587;
   1:  PR[91,3] = PR[90,3] + 13.439;
   1:L PR[91] R[100]mm/sec CNT100;
   1:  PR[91,1] = PR[90,1] + 18.006;
   1:  PR[91,2] = PR[90,2] + -16.644;
   1:  PR[91,3] = PR[90,3] + 13.445;
   1:L PR[91] R[100]mm/sec CNT100;
   1:  PR[91,1] = PR[90,1] + 18.498;
   1:  PR[91,2] = PR[90,2] + -16.653;
   1:  PR[91,3] = PR[90,3] + 13.451;
   1:L PR[91] R[100]mm/sec CNT100;
   1:  PR[91,1] = PR[90,1] + 18.878;
   1:  PR[91,2] = PR[90,2] + -16.658;
   1:  PR[91,3] = PR[90,3] + 13.454;
   1:L PR[91] R[100]mm/sec CNT100;
   1:  PR[91,1] = PR[90,1] + 19.751;
   1:  PR[91,2] = PR[90,2] + -16.630;
   1:  PR[91,3] = PR[90,3] + 13.456;
   1:L PR[91] R[100]mm/sec CNT100;
   1:  PR[91,1] = PR[90,1] + 20.619;
   1:  PR[91,2] = PR[90,2] + -16.559;
   1:  PR[91,3] = PR[90,3] + 13.462;
   1:L PR[91] R[100]mm/sec CNT100;
   1:  PR[91,1] = PR[90,1] + 21.481;
   1:  PR[91,2] = PR[90,2] + -16.447;
   1:  PR[91,3] = PR[90,3] + 13.468;
   1:L PR[91] R[100]mm/sec CNT100;
   1:  PR[91,1] = PR[90,1] + 22.334;
   1:  PR[91,2] = PR[90,2] + -16.294;
   1:  PR[91,3] = PR[90,3] + 13.473;
   1:L PR[91] R[100]mm/sec CNT100;
   1:  PR[91,1] = PR[90,1] + 23.181;
   1:  PR[91,2] = PR[90,2] + -16.098;
   1:  PR[91,3] = PR[90,3] + 13.479;
   1:L PR[91] R[100]mm/sec CNT100;
   1:  PR[91,1] = PR[90,1] + 24.003;
   1:  PR[91,2] = PR[90,2] + -15.866;
   1:  PR[91,3] = PR[90,3] + 13.485;
   1:L PR[91] R[100]mm/sec CNT100;
   1:  PR[91,1] = PR[90,1] + 24.817;
   1:  PR[91,2] = PR[90,2] + -15.593;
   1:  PR[91,3] = PR[90,3] + 13.490;
   1:L PR[91] R[100]mm/sec CNT100;
   1:  PR[91,1] = PR[90,1] + 25.614;
   1:  PR[91,2] = PR[90,2] + -15.282;
   1:  PR[91,3] = PR[90,3] + 13.496;
   1:L PR[91] R[100]mm/sec CNT100;
   1:  PR[91,1] = PR[90,1] + 26.393;
   1:  PR[91,2] = PR[90,2] + -14.934;
   1:  PR[91,3] = PR[90,3] + 13.502;
   1:L PR[91] R[100]mm/sec CNT100;
   1:  PR[91,1] = PR[90,1] + 27.153;
   1:  PR[91,2] = PR[90,2] + -14.550;
   1:  PR[91,3] = PR[90,3] + 13.507;
   1:L PR[91] R[100]mm/sec CNT100;
   1:  PR[91,1] = PR[90,1] + 27.892;
   1:  PR[91,2] = PR[90,2] + -14.130;
   1:  PR[91,3] = PR[90,3] + 13.513;
   1:L PR[91] R[100]mm/sec CNT100;
   1:  PR[91,1] = PR[90,1] + 28.607;
   1:  PR[91,2] = PR[90,2] + -13.676;
   1:  PR[91,3] = PR[90,3] + 13.518;
   1:L PR[91] R[100]mm/sec CNT100;
   1:  PR[91,1] = PR[90,1] + 29.298;
   1:  PR[91,2] = PR[90,2] + -13.189;
   1:  PR[91,3] = PR[90,3] + 13.524;
   1:L PR[91] R[100]mm/sec CNT100;
   1:  PR[91,1] = PR[90,1] + 29.963;
   1:  PR[91,2] = PR[90,2] + -12.670;
   1:  PR[91,3] = PR[90,3] + 13.529;
   1:L PR[91] R[100]mm/sec CNT100;
   1:  PR[91,1] = PR[90,1] + 30.601;
   1:  PR[91,2] = PR[90,2] + -12.120;
   1:  PR[91,3] = PR[90,3] + 13.535;
   1:L PR[91] R[100]mm/sec CNT100;
   1:  PR[91,1] = PR[90,1] + 31.210;
   1:  PR[91,2] = PR[90,2] + -11.540;
   1:  PR[91,3] = PR[90,3] + 13.540;
   1:L PR[91] R[100]mm/sec CNT100;
   1:  PR[91,1] = PR[90,1] + 31.789;
   1:  PR[91,2] = PR[90,2] + -10.931;
   1:  PR[91,3] = PR[90,3] + 13.546;
   1:L PR[91] R[100]mm/sec CNT100;
